LIN {X 0,Y 362.168,Z 797.832,A -85,B 0,C 180,E1 19612.506,E2 19612.506} C_VEL
LIN {X 0,Y 361.536,Z 796.314,A -85,B 0,C 180,E1 19613.999,E2 19613.999} C_VEL
LIN {X 0,Y 362.249,Z 796.809,A -85,B 0,C 180,E1 19623.883,E2 19623.883} C_VEL
LIN {X 0,Y 364.945,Z 802.489,A -85,B 0,C 180,E1 19627.878,E2 19627.878} C_VEL
LIN {X 0,Y 367.758,Z 805.063,A -85,B 0,C 180,E1 19630.43,E2 19630.43} C_VEL
LIN {X 0,Y 371.88,Z 810.734,A -85,B 0,C 180,E1 19633.506,E2 19633.506} C_VEL
LIN {X 0,Y 378.981,Z 821.207,A -85,B 0,C 180,E1 19637.693,E2 19637.693} C_VEL
LIN {X 0,Y 387.023,Z 832.702,A -85,B 0,C 180,E1 19641.464,E2 19641.464} C_VEL
LIN {X 0,Y 400.18,Z 854.108,A -85,B 0,C 180,E1 19646.784,E2 19646.784} C_VEL
LIN {X 0,Y 413.065,Z 880.296,A -85,B 0,C 180,E1 19651.645,E2 19651.645} C_VEL
LIN {X 0,Y 424.289,Z 910.677,A -85,B 0,C 180,E1 19656.18,E2 19656.18} C_VEL
LIN {X 0,Y 427.692,Z 923.118,A -85,B 0,C 180,E1 19657.818,E2 19657.818} C_VEL
LIN {X 0,Y 416.23,Z 964.506,A -85,B 0,C 180,E1 19660.322,E2 19660.322} C_VEL
LIN {X 0,Y 402.461,Z 1004.663,A -85,B 0,C 180,E1 19663.773,E2 19663.773} C_VEL
LIN {X 0,Y 388.693,Z 1040.022,A -85,B 0,C 180,E1 19668.003,E2 19668.003} C_VEL
LIN {X 0,Y 376.09,Z 1070.375,A -85,B 0,C 180,E1 19672.936,E2 19672.936} C_VEL
LIN {X 0,Y 364.901,Z 1097.162,A -85,B 0,C 180,E1 19678.824,E2 19678.824} C_VEL
LIN {X 0,Y 356.118,Z 1120.424,A -85,B 0,C 180,E1 19685.992,E2 19685.992} C_VEL
LIN {X 0,Y 351.388,Z 1136.328,A -85,B 0,C 180,E1 19693.124,E2 19693.124} C_VEL
LIN {X 0,Y 349.542,Z 1146.309,A -85,B 0,C 180,E1 19700.041,E2 19700.041} C_VEL
LIN {X 0,Y 349.172,Z 1150.432,A -85,B 0,C 180,E1 19705.033,E2 19705.033} C_VEL
LIN {X 0,Y 349.406,Z 1151.895,A -85,B 0,C 180,E1 19709.999,E2 19709.999} C_VEL
LIN {X 0,Y 349.323,Z 1149.313,A -85,B 0,C 180,E1 19717.455,E2 19717.455} C_VEL
LIN {X 0,Y 350.482,Z 1142.163,A -85,B 0,C 180,E1 19724.247,E2 19724.247} C_VEL
LIN {X 0,Y 354.503,Z 1128.114,A -85,B 0,C 180,E1 19731.898,E2 19731.898} C_VEL
LIN {X 0,Y 361.902,Z 1109.331,A -85,B 0,C 180,E1 19738.761,E2 19738.761} C_VEL
LIN {X 0,Y 372.688,Z 1085.078,A -85,B 0,C 180,E1 19745.117,E2 19745.117} C_VEL
LIN {X 0,Y 386.556,Z 1054.958,A -85,B 0,C 180,E1 19750.804,E2 19750.804} C_VEL
LIN {X 0,Y 401.988,Z 1019.714,A -85,B 0,C 180,E1 19755.578,E2 19755.578} C_VEL
LIN {X 0,Y 417.133,Z 980.614,A -85,B 0,C 180,E1 19759.349,E2 19759.349} C_VEL
LIN {X 0,Y 430.035,Z 940.71,A -85,B 0,C 180,E1 19762.083,E2 19762.083} C_VEL
LIN {X 0,Y 433.845,Z 925.859,A -85,B 0,C 180,E1 19762.938,E2 19762.938} C_VEL
LIN {X 0,Y 427.893,Z 906.219,A -85,B 0,C 180,E1 19765.929,E2 19765.929} C_VEL
LIN {X 0,Y 423.575,Z 900.256,A -85,B 0,C 180,E1 19767.396,E2 19767.396} C_VEL
LIN {X 0,Y 415.692,Z 891.837,A -85,B 0,C 180,E1 19769.971,E2 19769.971} C_VEL
LIN {X 0,Y 405.005,Z 869.047,A -85,B 0,C 180,E1 19775.094,E2 19775.094} C_VEL
LIN {X 0,Y 395.69,Z 852.613,A -85,B 0,C 180,E1 19780.05,E2 19780.05} C_VEL
LIN {X 0,Y 388.376,Z 840.695,A -85,B 0,C 180,E1 19784.924,E2 19784.924} C_VEL
LIN {X 0,Y 384.106,Z 833.994,A -85,B 0,C 180,E1 19788.805,E2 19788.805} C_VEL
LIN {X 0,Y 380.965,Z 827.944,A -85,B 0,C 180,E1 19793.437,E2 19793.437} C_VEL
LIN {X 0,Y 380.133,Z 827.154,A -85,B 0,C 180,E1 19802.281,E2 19802.281} C_VEL
LIN {X 0,Y 381.144,Z 828.782,A -85,B 0,C 180,E1 19804.693,E2 19804.693} C_VEL
LIN {X 0,Y 385.399,Z 836.304,A -85,B 0,C 180,E1 19810.307,E2 19810.307} C_VEL
LIN {X 0,Y 389.991,Z 844.13,A -85,B 0,C 180,E1 19814.191,E2 19814.191} C_VEL
LIN {X 0,Y 396.416,Z 855.261,A -85,B 0,C 180,E1 19818.472,E2 19818.472} C_VEL
LIN {X 0,Y 405.022,Z 872,A -85,B 0,C 180,E1 19823.353,E2 19823.353} C_VEL
LIN {X 0,Y 414.582,Z 895.457,A -85,B 0,C 180,E1 19828.579,E2 19828.579} C_VEL
LIN {X 0,Y 422.183,Z 920.876,A -85,B 0,C 180,E1 19833.177,E2 19833.177} C_VEL
LIN {X 0,Y 424.149,Z 932.657,A -85,B 0,C 180,E1 19834.976,E2 19834.976} C_VEL
LIN {X 0,Y 410.073,Z 973.06,A -85,B 0,C 180,E1 19838.101,E2 19838.101} C_VEL
LIN {X 0,Y 394.408,Z 1010.708,A -85,B 0,C 180,E1 19842.231,E2 19842.231} C_VEL
LIN {X 0,Y 379.532,Z 1042.173,A -85,B 0,C 180,E1 19847.015,E2 19847.015} C_VEL
LIN {X 0,Y 366.399,Z 1068.593,A -85,B 0,C 180,E1 19852.534,E2 19852.534} C_VEL
LIN {X 0,Y 354.767,Z 1091.747,A -85,B 0,C 180,E1 19859.262,E2 19859.262} C_VEL
LIN {X 0,Y 346.87,Z 1109.654,A -85,B 0,C 180,E1 19866.918,E2 19866.918} C_VEL
LIN {X 0,Y 342.767,Z 1121.009,A -85,B 0,C 180,E1 19874.663,E2 19874.663} C_VEL
LIN {X 0,Y 341.278,Z 1126.553,A -85,B 0,C 180,E1 19882.368,E2 19882.368} C_VEL
LIN {X 0,Y 341.472,Z 1126.707,A -85,B 0,C 180,E1 19890.001,E2 19890.001} C_VEL
LIN {X 0,Y 342.066,Z 1122.521,A -85,B 0,C 180,E1 19896.548,E2 19896.548} C_VEL
LIN {X 0,Y 344.669,Z 1112.858,A -85,B 0,C 180,E1 19903.955,E2 19903.955} C_VEL
LIN {X 0,Y 350.349,Z 1097.245,A -85,B 0,C 180,E1 19911.397,E2 19911.397} C_VEL
LIN {X 0,Y 360.014,Z 1075.116,A -85,B 0,C 180,E1 19918.521,E2 19918.521} C_VEL
LIN {X 0,Y 373.042,Z 1046.772,A -85,B 0,C 180,E1 19924.903,E2 19924.903} C_VEL
LIN {X 0,Y 387.331,Z 1014.182,A -85,B 0,C 180,E1 19930.139,E2 19930.139} C_VEL
LIN {X 0,Y 401.157,Z 979.377,A -85,B 0,C 180,E1 19934.184,E2 19934.184} C_VEL
LIN {X 0,Y 413.904,Z 941.564,A -85,B 0,C 180,E1 19937.419,E2 19937.419} C_VEL
LIN {X 0,Y 417.932,Z 926.539,A -85,B 0,C 180,E1 19938.504,E2 19938.504} C_VEL
LIN {X 0,Y 410.386,Z 897.331,A -85,B 0,C 180,E1 19942.987,E2 19942.987} C_VEL
LIN {X 0,Y 400.227,Z 871.059,A -85,B 0,C 180,E1 19947.767,E2 19947.767} C_VEL
LIN {X 0,Y 388.953,Z 848.616,A -85,B 0,C 180,E1 19952.842,E2 19952.842} C_VEL
LIN {X 0,Y 378.74,Z 831.473,A -85,B 0,C 180,E1 19957.951,E2 19957.951} C_VEL
LIN {X 0,Y 369.947,Z 818.286,A -85,B 0,C 180,E1 19963.385,E2 19963.385} C_VEL
LIN {X 0,Y 365.888,Z 812.166,A -85,B 0,C 180,E1 19966.717,E2 19966.717} C_VEL
LIN {X 0,Y 361.027,Z 805.323,A -85,B 0,C 180,E1 19972.86,E2 19972.86} C_VEL
LIN {X 0,Y 360.12,Z 803.979,A -85,B 0,C 180,E1 19975.183,E2 19975.183} C_VEL
LIN {X 0,Y 361.146,Z 804.69,A -85,B 0,C 180,E1 19983.669,E2 19983.669} C_VEL
LIN {X 0,Y 364.275,Z 810.621,A -85,B 0,C 180,E1 19988.193,E2 19988.193} C_VEL
LIN {X 0,Y 366.418,Z 812.851,A -85,B 0,C 180,E1 19990.164,E2 19990.164} C_VEL
LIN {X 0,Y 371.827,Z 820.887,A -85,B 0,C 180,E1 19994.257,E2 19994.257} C_VEL
LIN {X 0,Y 377.543,Z 829.283,A -85,B 0,C 180,E1 19997.612,E2 19997.612} C_VEL
LIN {X 0,Y 385.804,Z 841.914,A -85,B 0,C 180,E1 20001.686,E2 20001.686} C_VEL
LIN {X 0,Y 397.536,Z 862.222,A -85,B 0,C 180,E1 20006.672,E2 20006.672} C_VEL
LIN {X 0,Y 408.791,Z 885.918,A -85,B 0,C 180,E1 20011.156,E2 20011.156} C_VEL
LIN {X 0,Y 419.34,Z 916.182,A -85,B 0,C 180,E1 20015.795,E2 20015.795} C_VEL
LIN {X 0,Y 421.555,Z 927.264,A -85,B 0,C 180,E1 20017.21,E2 20017.21} C_VEL
LIN {X 0,Y 410.01,Z 967.1,A -85,B 0,C 180,E1 20019.709,E2 20019.709} C_VEL
LIN {X 0,Y 396.083,Z 1006.299,A -85,B 0,C 180,E1 20023.142,E2 20023.142} C_VEL
LIN {X 0,Y 381.298,Z 1042.819,A -85,B 0,C 180,E1 20027.643,E2 20027.643} C_VEL
LIN {X 0,Y 367.774,Z 1073.95,A -85,B 0,C 180,E1 20032.952,E2 20032.952} C_VEL
LIN {X 0,Y 356.83,Z 1099.215,A -85,B 0,C 180,E1 20038.821,E2 20038.821} C_VEL
LIN {X 0,Y 348.628,Z 1120.215,A -85,B 0,C 180,E1 20045.507,E2 20045.507} C_VEL
LIN {X 0,Y 343.368,Z 1137.166,A -85,B 0,C 180,E1 20053.377,E2 20053.377} C_VEL
LIN {X 0,Y 341.653,Z 1145.995,A -85,B 0,C 180,E1 20059.808,E2 20059.808} C_VEL
LIN {X 0,Y 341.284,Z 1150.137,A -85,B 0,C 180,E1 20064.918,E2 20064.918} C_VEL
LIN {X 0,Y 341.507,Z 1151.61,A -85,B 0,C 180,E1 20069.999,E2 20069.999} C_VEL
LIN {X 0,Y 341.426,Z 1149.049,A -85,B 0,C 180,E1 20077.629,E2 20077.629} C_VEL
LIN {X 0,Y 342.51,Z 1142.66,A -85,B 0,C 180,E1 20083.981,E2 20083.981} C_VEL
LIN {X 0,Y 345.94,Z 1130.613,A -85,B 0,C 180,E1 20091.121,E2 20091.121} C_VEL
LIN {X 0,Y 353.398,Z 1112.237,A -85,B 0,C 180,E1 20098.42,E2 20098.42} C_VEL
LIN {X 0,Y 365.132,Z 1086.928,A -85,B 0,C 180,E1 20105.406,E2 20105.406} C_VEL
LIN {X 0,Y 380.108,Z 1055.581,A -85,B 0,C 180,E1 20111.488,E2 20111.488} C_VEL
LIN {X 0,Y 396.368,Z 1019.642,A -85,B 0,C 180,E1 20116.413,E2 20116.413} C_VEL
LIN {X 0,Y 412.043,Z 980.377,A -85,B 0,C 180,E1 20120.214,E2 20120.214} C_VEL
LIN {X 0,Y 425.19,Z 940.845,A -85,B 0,C 180,E1 20122.925,E2 20122.925} C_VEL
LIN {X 0,Y 428.283,Z 929.273,A -85,B 0,C 180,E1 20123.606,E2 20123.606} C_VEL
LIN {X 0,Y 420.043,Z 902.49,A -85,B 0,C 180,E1 20127.962,E2 20127.962} C_VEL
LIN {X 0,Y 415.692,Z 891.837,A -85,B 0,C 180,E1 20129.971,E2 20129.971} C_VEL
LIN {X 0,Y 411.436,Z 886.846,A -85,B 0,C 180,E1 20131.549,E2 20131.549} C_VEL
LIN {X 0,Y 404.486,Z 881.278,A -85,B 0,C 180,E1 20134.056,E2 20134.056} C_VEL
LIN {X 0,Y 403.94,Z 880.243,A -85,B 0,C 180,E1 20134.322,E2 20134.322} C_VEL
LIN {X 0,Y 393.864,Z 860.717,A -85,B 0,C 180,E1 20139.954,E2 20139.954} C_VEL
LIN {X 0,Y 386.147,Z 847.843,A -85,B 0,C 180,E1 20145.415,E2 20145.415} C_VEL
LIN {X 0,Y 382.343,Z 841.592,A -85,B 0,C 180,E1 20149.041,E2 20149.041} C_VEL
LIN {X 0,Y 378.986,Z 835.151,A -85,B 0,C 180,E1 20154.64,E2 20154.64} C_VEL
LIN {X 0,Y 379.367,Z 835.251,A -85,B 0,C 180,E1 20163.857,E2 20163.857} C_VEL
LIN {X 0,Y 382.515,Z 841.74,A -85,B 0,C 180,E1 20168.879,E2 20168.879} C_VEL
LIN {X 0,Y 387.602,Z 851.333,A -85,B 0,C 180,E1 20173.863,E2 20173.863} C_VEL
LIN {X 0,Y 393.503,Z 862.183,A -85,B 0,C 180,E1 20178.108,E2 20178.108} C_VEL
LIN {X 0,Y 401.875,Z 879.654,A -85,B 0,C 180,E1 20183.254,E2 20183.254} C_VEL
LIN {X 0,Y 410.458,Z 901.841,A -85,B 0,C 180,E1 20188.263,E2 20188.263} C_VEL
LIN {X 0,Y 417.611,Z 928.524,A -85,B 0,C 180,E1 20193.179,E2 20193.179} C_VEL
LIN {X 0,Y 418.331,Z 936.224,A -85,B 0,C 180,E1 20194.321,E2 20194.321} C_VEL
LIN {X 0,Y 404.003,Z 975.78,A -85,B 0,C 180,E1 20197.458,E2 20197.458} C_VEL
LIN {X 0,Y 388.289,Z 1012.281,A -85,B 0,C 180,E1 20201.538,E2 20201.538} C_VEL
LIN {X 0,Y 372.079,Z 1045.221,A -85,B 0,C 180,E1 20206.684,E2 20206.684} C_VEL
LIN {X 0,Y 357.973,Z 1072.305,A -85,B 0,C 180,E1 20212.643,E2 20212.643} C_VEL
LIN {X 0,Y 346.862,Z 1093.638,A -85,B 0,C 180,E1 20219.212,E2 20219.212} C_VEL
LIN {X 0,Y 339.389,Z 1109.871,A -85,B 0,C 180,E1 20226.379,E2 20226.379} C_VEL
LIN {X 0,Y 334.988,Z 1121.246,A -85,B 0,C 180,E1 20234.298,E2 20234.298} C_VEL
LIN {X 0,Y 333.385,Z 1126.82,A -85,B 0,C 180,E1 20242.186,E2 20242.186} C_VEL
LIN {X 0,Y 333.328,Z 1127.532,A -85,B 0,C 180,E1 20247.403,E2 20247.403} C_VEL
LIN {X 0,Y 333.695,Z 1125.898,A -85,B 0,C 180,E1 20252.597,E2 20252.597} C_VEL
LIN {X 0,Y 334.796,Z 1120.388,A -85,B 0,C 180,E1 20259.091,E2 20259.091} C_VEL
LIN {X 0,Y 338.283,Z 1109.482,A -85,B 0,C 180,E1 20266.443,E2 20266.443} C_VEL
LIN {X 0,Y 345.277,Z 1092.289,A -85,B 0,C 180,E1 20273.882,E2 20273.882} C_VEL
LIN {X 0,Y 355.746,Z 1069.725,A -85,B 0,C 180,E1 20280.647,E2 20280.647} C_VEL
LIN {X 0,Y 368.456,Z 1043,A -85,B 0,C 180,E1 20286.402,E2 20286.402} C_VEL
LIN {X 0,Y 383.057,Z 1010.649,A -85,B 0,C 180,E1 20291.457,E2 20291.457} C_VEL
LIN {X 0,Y 397.955,Z 973.716,A -85,B 0,C 180,E1 20295.603,E2 20295.603} C_VEL
LIN {X 0,Y 411.711,Z 932.607,A -85,B 0,C 180,E1 20298.891,E2 20298.891} C_VEL
LIN {X 0,Y 411.505,Z 926.566,A -85,B 0,C 180,E1 20299.627,E2 20299.627} C_VEL
LIN {X 0,Y 404.09,Z 897.94,A -85,B 0,C 180,E1 20304.243,E2 20304.243} C_VEL
LIN {X 0,Y 393.436,Z 870.633,A -85,B 0,C 180,E1 20309.569,E2 20309.569} C_VEL
LIN {X 0,Y 382.417,Z 849.153,A -85,B 0,C 180,E1 20314.976,E2 20314.976} C_VEL
LIN {X 0,Y 374.275,Z 835.712,A -85,B 0,C 180,E1 20319.516,E2 20319.516} C_VEL
LIN {X 0,Y 367.793,Z 825.425,A -85,B 0,C 180,E1 20324.031,E2 20324.031} C_VEL
LIN {X 0,Y 363.665,Z 818.969,A -85,B 0,C 180,E1 20327.703,E2 20327.703} C_VEL
LIN {X 0,Y 359.883,Z 812.953,A -85,B 0,C 180,E1 20333.14,E2 20333.14} C_VEL
LIN {X 0,Y 358.713,Z 811.507,A -85,B 0,C 180,E1 20337.582,E2 20337.582} C_VEL
LIN {X 0,Y 360.103,Z 812.832,A -85,B 0,C 180,E1 20343.605,E2 20343.605} C_VEL
LIN {X 0,Y 363.845,Z 818.876,A -85,B 0,C 180,E1 20348.804,E2 20348.804} C_VEL
LIN {X 0,Y 370.025,Z 828.147,A -85,B 0,C 180,E1 20353.876,E2 20353.876} C_VEL
LIN {X 0,Y 378.227,Z 840.611,A -85,B 0,C 180,E1 20358.784,E2 20358.784} C_VEL
LIN {X 0,Y 389.385,Z 859.782,A -85,B 0,C 180,E1 20364.191,E2 20364.191} C_VEL
LIN {X 0,Y 401.157,Z 883.666,A -85,B 0,C 180,E1 20369.264,E2 20369.264} C_VEL
LIN {X 0,Y 411.593,Z 912.314,A -85,B 0,C 180,E1 20374.037,E2 20374.037} C_VEL
LIN {X 0,Y 415.852,Z 929.747,A -85,B 0,C 180,E1 20376.488,E2 20376.488} C_VEL
LIN {X 0,Y 403.786,Z 969.68,A -85,B 0,C 180,E1 20379.07,E2 20379.07} C_VEL
LIN {X 0,Y 389.596,Z 1008.144,A -85,B 0,C 180,E1 20382.527,E2 20382.527} C_VEL
LIN {X 0,Y 374.466,Z 1044.278,A -85,B 0,C 180,E1 20387.079,E2 20387.079} C_VEL
LIN {X 0,Y 359.392,Z 1077.666,A -85,B 0,C 180,E1 20393.004,E2 20393.004} C_VEL
LIN {X 0,Y 347.197,Z 1104.998,A -85,B 0,C 180,E1 20399.885,E2 20399.885} C_VEL
LIN {X 0,Y 338.739,Z 1126.558,A -85,B 0,C 180,E1 20407.715,E2 20407.715} C_VEL
LIN {X 0,Y 334.81,Z 1139.995,A -85,B 0,C 180,E1 20415.035,E2 20415.035} C_VEL
LIN {X 0,Y 333.546,Z 1148.087,A -85,B 0,C 180,E1 20422.187,E2 20422.187} C_VEL
LIN {X 0,Y 333.435,Z 1150.905,A -85,B 0,C 180,E1 20427.401,E2 20427.401} C_VEL
LIN {X 0,Y 333.404,Z 1151.1,A -85,B 0,C 180,E1 20432.596,E2 20432.596} C_VEL
LIN {X 0,Y 333.647,Z 1147.89,A -85,B 0,C 180,E1 20439.119,E2 20439.119} C_VEL
LIN {X 0,Y 335.145,Z 1140.554,A -85,B 0,C 180,E1 20445.694,E2 20445.694} C_VEL
LIN {X 0,Y 340.055,Z 1126.288,A -85,B 0,C 180,E1 20453.572,E2 20453.572} C_VEL
LIN {X 0,Y 349.349,Z 1105.179,A -85,B 0,C 180,E1 20461.267,E2 20461.267} C_VEL
LIN {X 0,Y 363.057,Z 1077.643,A -85,B 0,C 180,E1 20468.187,E2 20468.187} C_VEL
LIN {X 0,Y 379.117,Z 1044.881,A -85,B 0,C 180,E1 20473.963,E2 20473.963} C_VEL
LIN {X 0,Y 395.082,Z 1009.645,A -85,B 0,C 180,E1 20478.364,E2 20478.364} C_VEL
LIN {X 0,Y 409.577,Z 973.339,A -85,B 0,C 180,E1 20481.627,E2 20481.627} C_VEL
LIN {X 0,Y 422.829,Z 932.79,A -85,B 0,C 180,E1 20484.272,E2 20484.272} C_VEL
LIN {X 0,Y 414.989,Z 906.692,A -85,B 0,C 180,E1 20488.677,E2 20488.677} C_VEL
LIN {X 0,Y 404.705,Z 881.627,A -85,B 0,C 180,E1 20493.956,E2 20493.956} C_VEL
LIN {X 0,Y 403.94,Z 880.243,A -85,B 0,C 180,E1 20494.322,E2 20494.322} C_VEL
LIN {X 0,Y 400.075,Z 875.927,A -85,B 0,C 180,E1 20495.995,E2 20495.995} C_VEL
LIN {X 0,Y 393.13,Z 871.803,A -85,B 0,C 180,E1 20498.985,E2 20498.985} C_VEL
LIN {X 0,Y 384.724,Z 856.032,A -85,B 0,C 180,E1 20505.069,E2 20505.069} C_VEL
LIN {X 0,Y 380.382,Z 849.039,A -85,B 0,C 180,E1 20509.418,E2 20509.418} C_VEL
LIN {X 0,Y 377.669,Z 842.974,A -85,B 0,C 180,E1 20514.264,E2 20514.264} C_VEL
LIN {X 0,Y 377.788,Z 843.047,A -85,B 0,C 180,E1 20523.73,E2 20523.73} C_VEL
LIN {X 0,Y 380.727,Z 849.492,A -85,B 0,C 180,E1 20528.921,E2 20528.921} C_VEL
LIN {X 0,Y 387.257,Z 861.984,A -85,B 0,C 180,E1 20535.2,E2 20535.2} C_VEL
LIN {X 0,Y 395.349,Z 879.25,A -85,B 0,C 180,E1 20540.998,E2 20540.998} C_VEL
LIN {X 0,Y 403.722,Z 900.712,A -85,B 0,C 180,E1 20546.359,E2 20546.359} C_VEL
LIN {X 0,Y 410.328,Z 923.987,A -85,B 0,C 180,E1 20551.034,E2 20551.034} C_VEL
LIN {X 0,Y 412.849,Z 938.974,A -85,B 0,C 180,E1 20553.592,E2 20553.592} C_VEL
LIN {X 0,Y 398.879,Z 976.352,A -85,B 0,C 180,E1 20556.595,E2 20556.595} C_VEL
LIN {X 0,Y 382.928,Z 1012.308,A -85,B 0,C 180,E1 20560.624,E2 20560.624} C_VEL
LIN {X 0,Y 366.202,Z 1045.309,A -85,B 0,C 180,E1 20565.81,E2 20565.81} C_VEL
LIN {X 0,Y 352.17,Z 1071.253,A -85,B 0,C 180,E1 20571.527,E2 20571.527} C_VEL
LIN {X 0,Y 340.775,Z 1092.108,A -85,B 0,C 180,E1 20577.853,E2 20577.853} C_VEL
LIN {X 0,Y 331.938,Z 1110.085,A -85,B 0,C 180,E1 20585.815,E2 20585.815} C_VEL
LIN {X 0,Y 327.249,Z 1121.482,A -85,B 0,C 180,E1 20593.917,E2 20593.917} C_VEL
LIN {X 0,Y 325.493,Z 1127.087,A -85,B 0,C 180,E1 20601.996,E2 20601.996} C_VEL
LIN {X 0,Y 325.43,Z 1127.819,A -85,B 0,C 180,E1 20607.34,E2 20607.34} C_VEL
LIN {X 0,Y 325.813,Z 1126.206,A -85,B 0,C 180,E1 20612.66,E2 20612.66} C_VEL
LIN {X 0,Y 326.97,Z 1120.719,A -85,B 0,C 180,E1 20619.31,E2 20619.31} C_VEL
LIN {X 0,Y 330.453,Z 1110.344,A -85,B 0,C 180,E1 20626.539,E2 20626.539} C_VEL
LIN {X 0,Y 337.172,Z 1094.37,A -85,B 0,C 180,E1 20633.79,E2 20633.79} C_VEL
LIN {X 0,Y 347.161,Z 1073.675,A -85,B 0,C 180,E1 20640.4,E2 20640.4} C_VEL
LIN {X 0,Y 360.579,Z 1046.711,A -85,B 0,C 180,E1 20646.552,E2 20646.552} C_VEL
LIN {X 0,Y 376.254,Z 1013.188,A -85,B 0,C 180,E1 20651.994,E2 20651.994} C_VEL
LIN {X 0,Y 391.949,Z 975.567,A -85,B 0,C 180,E1 20656.306,E2 20656.306} C_VEL
LIN {X 0,Y 405.592,Z 936.216,A -85,B 0,C 180,E1 20659.533,E2 20659.533} C_VEL
LIN {X 0,Y 405.888,Z 930.287,A -85,B 0,C 180,E1 20660.23,E2 20660.23} C_VEL
LIN {X 0,Y 399.275,Z 903.126,A -85,B 0,C 180,E1 20664.752,E2 20664.752} C_VEL
LIN {X 0,Y 389.421,Z 876.566,A -85,B 0,C 180,E1 20670.061,E2 20670.061} C_VEL
LIN {X 0,Y 379.183,Z 855.426,A -85,B 0,C 180,E1 20675.554,E2 20675.554} C_VEL
LIN {X 0,Y 370.32,Z 839.719,A -85,B 0,C 180,E1 20681.027,E2 20681.027} C_VEL
LIN {X 0,Y 365.445,Z 832.455,A -85,B 0,C 180,E1 20684.65,E2 20684.65} C_VEL
LIN {X 0,Y 361.967,Z 826.507,A -85,B 0,C 180,E1 20688.205,E2 20688.205} C_VEL
LIN {X 0,Y 358.567,Z 820.126,A -85,B 0,C 180,E1 20693.646,E2 20693.646} C_VEL
LIN {X 0,Y 358.803,Z 820.091,A -85,B 0,C 180,E1 20703.164,E2 20703.164} C_VEL
LIN {X 0,Y 362.094,Z 826.331,A -85,B 0,C 180,E1 20708.243,E2 20708.243} C_VEL
LIN {X 0,Y 363.768,Z 828.917,A -85,B 0,C 180,E1 20709.937,E2 20709.937} C_VEL
LIN {X 0,Y 368.356,Z 835.989,A -85,B 0,C 180,E1 20713.713,E2 20713.713} C_VEL
LIN {X 0,Y 376.027,Z 848.137,A -85,B 0,C 180,E1 20718.518,E2 20718.518} C_VEL
LIN {X 0,Y 386.853,Z 867.538,A -85,B 0,C 180,E1 20724.054,E2 20724.054} C_VEL
LIN {X 0,Y 397.426,Z 890.611,A -85,B 0,C 180,E1 20729.01,E2 20729.01} C_VEL
LIN {X 0,Y 407.103,Z 919.151,A -85,B 0,C 180,E1 20733.823,E2 20733.823} C_VEL
LIN {X 0,Y 410.257,Z 931.658,A -85,B 0,C 180,E1 20735.696,E2 20735.696} C_VEL
LIN {X 0,Y 397.025,Z 973.907,A -85,B 0,C 180,E1 20738.536,E2 20738.536} C_VEL
LIN {X 0,Y 383.326,Z 1009.53,A -85,B 0,C 180,E1 20741.841,E2 20741.841} C_VEL
LIN {X 0,Y 368.52,Z 1043.8,A -85,B 0,C 180,E1 20746.213,E2 20746.213} C_VEL
LIN {X 0,Y 352.898,Z 1077.24,A -85,B 0,C 180,E1 20752.205,E2 20752.205} C_VEL
LIN {X 0,Y 340.007,Z 1104.835,A -85,B 0,C 180,E1 20759.261,E2 20759.261} C_VEL
LIN {X 0,Y 331.227,Z 1126.198,A -85,B 0,C 180,E1 20767.182,E2 20767.182} C_VEL
LIN {X 0,Y 326.845,Z 1140.502,A -85,B 0,C 180,E1 20775.242,E2 20775.242} C_VEL
LIN {X 0,Y 325.65,Z 1147.783,A -85,B 0,C 180,E1 20781.996,E2 20781.996} C_VEL
LIN {X 0,Y 325.529,Z 1150.612,A -85,B 0,C 180,E1 20787.338,E2 20787.338} C_VEL
LIN {X 0,Y 325.5,Z 1150.823,A -85,B 0,C 180,E1 20792.659,E2 20792.659} C_VEL
LIN {X 0,Y 325.785,Z 1147.626,A -85,B 0,C 180,E1 20799.341,E2 20799.341} C_VEL
LIN {X 0,Y 327.405,Z 1140.314,A -85,B 0,C 180,E1 20806.075,E2 20806.075} C_VEL
LIN {X 0,Y 332.593,Z 1126.067,A -85,B 0,C 180,E1 20814.135,E2 20814.135} C_VEL
LIN {X 0,Y 342.411,Z 1104.986,A -85,B 0,C 180,E1 20821.975,E2 20821.975} C_VEL
LIN {X 0,Y 356.059,Z 1078.611,A -85,B 0,C 180,E1 20828.748,E2 20828.748} C_VEL
LIN {X 0,Y 371.239,Z 1048.787,A -85,B 0,C 180,E1 20834.21,E2 20834.21} C_VEL
LIN {X 0,Y 387.036,Z 1015.824,A -85,B 0,C 180,E1 20838.564,E2 20838.564} C_VEL
LIN {X 0,Y 402.968,Z 977.945,A -85,B 0,C 180,E1 20842.168,E2 20842.168} C_VEL
LIN {X 0,Y 417.168,Z 935.697,A -85,B 0,C 180,E1 20845.043,E2 20845.043} C_VEL
LIN {X 0,Y 409.307,Z 908.802,A -85,B 0,C 180,E1 20849.81,E2 20849.81} C_VEL
LIN {X 0,Y 400.089,Z 885.921,A -85,B 0,C 180,E1 20854.924,E2 20854.924} C_VEL
LIN {X 0,Y 393.13,Z 871.803,A -85,B 0,C 180,E1 20858.985,E2 20858.985} C_VEL
LIN {X 0,Y 383.944,Z 866.755,A -85,B 0,C 180,E1 20863.942,E2 20863.942} C_VEL
LIN {X 0,Y 378.689,Z 856.9,A -85,B 0,C 180,E1 20869.225,E2 20869.225} C_VEL
LIN {X 0,Y 375.718,Z 850.567,A -85,B 0,C 180,E1 20874.812,E2 20874.812} C_VEL
LIN {X 0,Y 375.909,Z 850.766,A -85,B 0,C 180,E1 20883.604,E2 20883.604} C_VEL
LIN {X 0,Y 379.379,Z 859.105,A -85,B 0,C 180,E1 20889.748,E2 20889.748} C_VEL
LIN {X 0,Y 384.502,Z 869.078,A -85,B 0,C 180,E1 20894.874,E2 20894.874} C_VEL
LIN {X 0,Y 392.77,Z 888.014,A -85,B 0,C 180,E1 20901.219,E2 20901.219} C_VEL
LIN {X 0,Y 400.164,Z 908.969,A -85,B 0,C 180,E1 20906.476,E2 20906.476} C_VEL
LIN {X 0,Y 406.245,Z 933.446,A -85,B 0,C 180,E1 20911.381,E2 20911.381} C_VEL
LIN {X 0,Y 407.489,Z 941.696,A -85,B 0,C 180,E1 20912.85,E2 20912.85} C_VEL
LIN {X 0,Y 393.181,Z 978.428,A -85,B 0,C 180,E1 20915.853,E2 20915.853} C_VEL
LIN {X 0,Y 376.512,Z 1014.676,A -85,B 0,C 180,E1 20920,E2 20920} C_VEL
LIN {X 0,Y 359.419,Z 1047.186,A -85,B 0,C 180,E1 20925.228,E2 20925.228} C_VEL
LIN {X 0,Y 343.737,Z 1074.964,A -85,B 0,C 180,E1 20931.616,E2 20931.616} C_VEL
LIN {X 0,Y 331.918,Z 1095.712,A -85,B 0,C 180,E1 20938.431,E2 20938.431} C_VEL
LIN {X 0,Y 323.933,Z 1111.426,A -85,B 0,C 180,E1 20945.911,E2 20945.911} C_VEL
LIN {X 0,Y 319.493,Z 1121.72,A -85,B 0,C 180,E1 20953.516,E2 20953.516} C_VEL
LIN {X 0,Y 317.602,Z 1127.355,A -85,B 0,C 180,E1 20961.795,E2 20961.795} C_VEL
LIN {X 0,Y 317.549,Z 1128.047,A -85,B 0,C 180,E1 20967.732,E2 20967.732} C_VEL
LIN {X 0,Y 317.994,Z 1125.865,A -85,B 0,C 180,E1 20973.785,E2 20973.785} C_VEL
LIN {X 0,Y 319.578,Z 1119.538,A -85,B 0,C 180,E1 20980.904,E2 20980.904} C_VEL
LIN {X 0,Y 323.845,Z 1108.074,A -85,B 0,C 180,E1 20988.36,E2 20988.36} C_VEL
LIN {X 0,Y 331.552,Z 1091.372,A -85,B 0,C 180,E1 20995.658,E2 20995.658} C_VEL
LIN {X 0,Y 343.983,Z 1066.921,A -85,B 0,C 180,E1 21002.983,E2 21002.983} C_VEL
LIN {X 0,Y 359.118,Z 1037.325,A -85,B 0,C 180,E1 21009.138,E2 21009.138} C_VEL
LIN {X 0,Y 374.731,Z 1004.024,A -85,B 0,C 180,E1 21014.077,E2 21014.077} C_VEL
LIN {X 0,Y 389.608,Z 968.224,A -85,B 0,C 180,E1 21017.884,E2 21017.884} C_VEL
LIN {X 0,Y 400.512,Z 935.803,A -85,B 0,C 180,E1 21020.539,E2 21020.539} C_VEL
LIN {X 0,Y 394.377,Z 908.239,A -85,B 0,C 180,E1 21025.256,E2 21025.256} C_VEL
LIN {X 0,Y 385.437,Z 882.576,A -85,B 0,C 180,E1 21030.545,E2 21030.545} C_VEL
LIN {X 0,Y 376.01,Z 862.069,A -85,B 0,C 180,E1 21035.99,E2 21035.99} C_VEL
LIN {X 0,Y 367.793,Z 846.8,A -85,B 0,C 180,E1 21041.459,E2 21041.459} C_VEL
LIN {X 0,Y 363.39,Z 839.781,A -85,B 0,C 180,E1 21045.056,E2 21045.056} C_VEL
LIN {X 0,Y 360.048,Z 833.919,A -85,B 0,C 180,E1 21048.652,E2 21048.652} C_VEL
LIN {X 0,Y 357.095,Z 827.473,A -85,B 0,C 180,E1 21054.534,E2 21054.534} C_VEL
LIN {X 0,Y 357.586,Z 828.165,A -85,B 0,C 180,E1 21063.099,E2 21063.099} C_VEL
LIN {X 0,Y 361.265,Z 834.443,A -85,B 0,C 180,E1 21068.716,E2 21068.716} C_VEL
LIN {X 0,Y 366.619,Z 843.923,A -85,B 0,C 180,E1 21073.627,E2 21073.627} C_VEL
LIN {X 0,Y 373.705,Z 855.774,A -85,B 0,C 180,E1 21078.332,E2 21078.332} C_VEL
LIN {X 0,Y 383.997,Z 875.148,A -85,B 0,C 180,E1 21083.924,E2 21083.924} C_VEL
LIN {X 0,Y 394.603,Z 900.168,A -85,B 0,C 180,E1 21089.238,E2 21089.238} C_VEL
LIN {X 0,Y 403.088,Z 928.393,A -85,B 0,C 180,E1 21094.025,E2 21094.025} C_VEL
LIN {X 0,Y 404.362,Z 935.699,A -85,B 0,C 180,E1 21095.06,E2 21095.06} C_VEL
LIN {X 0,Y 390.477,Z 977.703,A -85,B 0,C 180,E1 21097.955,E2 21097.955} C_VEL
LIN {X 0,Y 374.936,Z 1016.114,A -85,B 0,C 180,E1 21101.724,E2 21101.724} C_VEL
LIN {X 0,Y 360.049,Z 1048.704,A -85,B 0,C 180,E1 21106.17,E2 21106.17} C_VEL
LIN {X 0,Y 345.317,Z 1078.975,A -85,B 0,C 180,E1 21111.861,E2 21111.861} C_VEL
LIN {X 0,Y 332.941,Z 1104.439,A -85,B 0,C 180,E1 21118.535,E2 21118.535} C_VEL
LIN {X 0,Y 323.711,Z 1125.836,A -85,B 0,C 180,E1 21126.621,E2 21126.621} C_VEL
LIN {X 0,Y 319.048,Z 1140.206,A -85,B 0,C 180,E1 21134.899,E2 21134.899} C_VEL
LIN {X 0,Y 317.774,Z 1147.48,A -85,B 0,C 180,E1 21141.797,E2 21141.797} C_VEL
LIN {X 0,Y 317.637,Z 1150.318,A -85,B 0,C 180,E1 21147.272,E2 21147.272} C_VEL
LIN {X 0,Y 317.614,Z 1150.546,A -85,B 0,C 180,E1 21152.725,E2 21152.725} C_VEL
LIN {X 0,Y 317.921,Z 1147.363,A -85,B 0,C 180,E1 21159.575,E2 21159.575} C_VEL
LIN {X 0,Y 319.648,Z 1140.073,A -85,B 0,C 180,E1 21166.476,E2 21166.476} C_VEL
LIN {X 0,Y 325.181,Z 1125.847,A -85,B 0,C 180,E1 21174.721,E2 21174.721} C_VEL
LIN {X 0,Y 335.486,Z 1104.791,A -85,B 0,C 180,E1 21182.716,E2 21182.716} C_VEL
LIN {X 0,Y 350.026,Z 1078.004,A -85,B 0,C 180,E1 21189.681,E2 21189.681} C_VEL
LIN {X 0,Y 365.95,Z 1047.779,A -85,B 0,C 180,E1 21195.235,E2 21195.235} C_VEL
LIN {X 0,Y 382.652,Z 1013.743,A -85,B 0,C 180,E1 21199.697,E2 21199.697} C_VEL
LIN {X 0,Y 398.699,Z 976.454,A -85,B 0,C 180,E1 21203.191,E2 21203.191} C_VEL
LIN {X 0,Y 411.66,Z 939.215,A -85,B 0,C 180,E1 21205.731,E2 21205.731} C_VEL
LIN {X 0,Y 404.8,Z 914.149,A -85,B 0,C 180,E1 21210.341,E2 21210.341} C_VEL
LIN {X 0,Y 395.753,Z 890.567,A -85,B 0,C 180,E1 21215.774,E2 21215.774} C_VEL
LIN {X 0,Y 387.603,Z 873.8,A -85,B 0,C 180,E1 21221.068,E2 21221.068} C_VEL
LIN {X 0,Y 383.944,Z 866.755,A -85,B 0,C 180,E1 21223.942,E2 21223.942} C_VEL
LIN {X 0,Y 381.372,Z 864.663,A -85,B 0,C 180,E1 21225.827,E2 21225.827} C_VEL
LIN {X 0,Y 376.903,Z 864.655,A -85,B 0,C 180,E1 21229.103,E2 21229.103} C_VEL
LIN {X 0,Y 373.882,Z 858.254,A -85,B 0,C 180,E1 21234.787,E2 21234.787} C_VEL
LIN {X 0,Y 373.989,Z 858.474,A -85,B 0,C 180,E1 21243.478,E2 21243.478} C_VEL
LIN {X 0,Y 377.041,Z 866.741,A -85,B 0,C 180,E1 21249.663,E2 21249.663} C_VEL
LIN {X 0,Y 381.445,Z 875.681,A -85,B 0,C 180,E1 21254.336,E2 21254.336} C_VEL
LIN {X 0,Y 388.611,Z 893.258,A -85,B 0,C 180,E1 21260.485,E2 21260.485} C_VEL
LIN {X 0,Y 395.385,Z 913.596,A -85,B 0,C 180,E1 21265.767,E2 21265.767} C_VEL
LIN {X 0,Y 400.908,Z 937.73,A -85,B 0,C 180,E1 21270.793,E2 21270.793} C_VEL
LIN {X 0,Y 401.54,Z 946.214,A -85,B 0,C 180,E1 21272.206,E2 21272.206} C_VEL
LIN {X 0,Y 385.131,Z 986.111,A -85,B 0,C 180,E1 21275.659,E2 21275.659} C_VEL
LIN {X 0,Y 368.597,Z 1019.893,A -85,B 0,C 180,E1 21279.767,E2 21279.767} C_VEL
LIN {X 0,Y 352.391,Z 1049.424,A -85,B 0,C 180,E1 21284.723,E2 21284.723} C_VEL
LIN {X 0,Y 336.663,Z 1076.283,A -85,B 0,C 180,E1 21291.071,E2 21291.071} C_VEL
LIN {X 0,Y 324.003,Z 1097.604,A -85,B 0,C 180,E1 21298.355,E2 21298.355} C_VEL
LIN {X 0,Y 315.734,Z 1113.1,A -85,B 0,C 180,E1 21306.221,E2 21306.221} C_VEL
LIN {X 0,Y 311.753,Z 1121.958,A -85,B 0,C 180,E1 21313.094,E2 21313.094} C_VEL
LIN {X 0,Y 310.111,Z 1126.345,A -85,B 0,C 180,E1 21318.762,E2 21318.762} C_VEL
LIN {X 0,Y 309.604,Z 1128.301,A -85,B 0,C 180,E1 21324.4,E2 21324.4} C_VEL
LIN {X 0,Y 309.907,Z 1127.894,A -85,B 0,C 180,E1 21330.002,E2 21330.002} C_VEL
LIN {X 0,Y 310.597,Z 1123.987,A -85,B 0,C 180,E1 21336.988,E2 21336.988} C_VEL
LIN {X 0,Y 313.61,Z 1114.945,A -85,B 0,C 180,E1 21344.941,E2 21344.941} C_VEL
LIN {X 0,Y 320.823,Z 1098.756,A -85,B 0,C 180,E1 21353.498,E2 21353.498} C_VEL
LIN {X 0,Y 332.857,Z 1075.713,A -85,B 0,C 180,E1 21361.473,E2 21361.473} C_VEL
LIN {X 0,Y 347.532,Z 1048.253,A -85,B 0,C 180,E1 21367.997,E2 21367.997} C_VEL
LIN {X 0,Y 363.178,Z 1017.074,A -85,B 0,C 180,E1 21373.255,E2 21373.255} C_VEL
LIN {X 0,Y 378.531,Z 983.123,A -85,B 0,C 180,E1 21377.377,E2 21377.377} C_VEL
LIN {X 0,Y 393.204,Z 944.516,A -85,B 0,C 180,E1 21380.789,E2 21380.789} C_VEL
LIN {X 0,Y 394.679,Z 938.576,A -85,B 0,C 180,E1 21381.308,E2 21381.308} C_VEL
LIN {X 0,Y 389.161,Z 912.175,A -85,B 0,C 180,E1 21386.002,E2 21386.002} C_VEL
LIN {X 0,Y 381.104,Z 887.648,A -85,B 0,C 180,E1 21391.258,E2 21391.258} C_VEL
LIN {X 0,Y 372.296,Z 867.626,A -85,B 0,C 180,E1 21396.767,E2 21396.767} C_VEL
LIN {X 0,Y 364.979,Z 853.542,A -85,B 0,C 180,E1 21402.069,E2 21402.069} C_VEL
LIN {X 0,Y 361.019,Z 846.766,A -85,B 0,C 180,E1 21405.606,E2 21405.606} C_VEL
LIN {X 0,Y 358.456,Z 841.641,A -85,B 0,C 180,E1 21408.736,E2 21408.736} C_VEL
LIN {X 0,Y 355.425,Z 835.16,A -85,B 0,C 180,E1 21415.119,E2 21415.119} C_VEL
LIN {X 0,Y 356.075,Z 835.968,A -85,B 0,C 180,E1 21422.96,E2 21422.96} C_VEL
LIN {X 0,Y 360.19,Z 843.854,A -85,B 0,C 180,E1 21429.351,E2 21429.351} C_VEL
LIN {X 0,Y 364.565,Z 851.493,A -85,B 0,C 180,E1 21433.4,E2 21433.4} C_VEL
LIN {X 0,Y 371.208,Z 863.164,A -85,B 0,C 180,E1 21438.076,E2 21438.076} C_VEL
LIN {X 0,Y 380.594,Z 881.85,A -85,B 0,C 180,E1 21443.533,E2 21443.533} C_VEL
LIN {X 0,Y 389.925,Z 905.205,A -85,B 0,C 180,E1 21448.649,E2 21448.649} C_VEL
LIN {X 0,Y 397.752,Z 932.489,A -85,B 0,C 180,E1 21453.415,E2 21453.415} C_VEL
LIN {X 0,Y 398.412,Z 939.292,A -85,B 0,C 180,E1 21454.36,E2 21454.36} C_VEL
LIN {X 0,Y 384.435,Z 979.974,A -85,B 0,C 180,E1 21457.251,E2 21457.251} C_VEL
LIN {X 0,Y 368.316,Z 1018.482,A -85,B 0,C 180,E1 21461.113,E2 21461.113} C_VEL
LIN {X 0,Y 351.615,Z 1053.61,A -85,B 0,C 180,E1 21466.136,E2 21466.136} C_VEL
LIN {X 0,Y 336.757,Z 1082.717,A -85,B 0,C 180,E1 21471.975,E2 21471.975} C_VEL
LIN {X 0,Y 324.972,Z 1106.056,A -85,B 0,C 180,E1 21478.456,E2 21478.456} C_VEL
LIN {X 0,Y 316.196,Z 1125.563,A -85,B 0,C 180,E1 21486.076,E2 21486.076} C_VEL
LIN {X 0,Y 311.273,Z 1139.873,A -85,B 0,C 180,E1 21494.512,E2 21494.512} C_VEL
LIN {X 0,Y 309.884,Z 1147.176,A -85,B 0,C 180,E1 21501.586,E2 21501.586} C_VEL
LIN {X 0,Y 309.759,Z 1150.025,A -85,B 0,C 180,E1 21507.202,E2 21507.202} C_VEL
LIN {X 0,Y 309.706,Z 1150.268,A -85,B 0,C 180,E1 21512.795,E2 21512.795} C_VEL
LIN {X 0,Y 310.035,Z 1147.098,A -85,B 0,C 180,E1 21519.82,E2 21519.82} C_VEL
LIN {X 0,Y 311.899,Z 1139.831,A -85,B 0,C 180,E1 21526.898,E2 21526.898} C_VEL
LIN {X 0,Y 317.95,Z 1125.332,A -85,B 0,C 180,E1 21535.475,E2 21535.475} C_VEL
LIN {X 0,Y 328.642,Z 1104.597,A -85,B 0,C 180,E1 21543.486,E2 21543.486} C_VEL
LIN {X 0,Y 343.542,Z 1078.284,A -85,B 0,C 180,E1 21550.449,E2 21550.449} C_VEL
LIN {X 0,Y 359.547,Z 1049.037,A -85,B 0,C 180,E1 21555.935,E2 21555.935} C_VEL
LIN {X 0,Y 376.428,Z 1015.993,A -85,B 0,C 180,E1 21560.374,E2 21560.374} C_VEL
LIN {X 0,Y 393.957,Z 976.48,A -85,B 0,C 180,E1 21564.122,E2 21564.122} C_VEL
LIN {X 0,Y 406.1,Z 942.36,A -85,B 0,C 180,E1 21566.511,E2 21566.511} C_VEL
LIN {X 0,Y 399.936,Z 918.55,A -85,B 0,C 180,E1 21571.063,E2 21571.063} C_VEL
LIN {X 0,Y 392.22,Z 897.181,A -85,B 0,C 180,E1 21576.146,E2 21576.146} C_VEL
LIN {X 0,Y 384.558,Z 880.476,A -85,B 0,C 180,E1 21581.54,E2 21581.54} C_VEL
LIN {X 0,Y 378.944,Z 869.522,A -85,B 0,C 180,E1 21586.477,E2 21586.477} C_VEL
LIN {X 0,Y 376.903,Z 864.655,A -85,B 0,C 180,E1 21589.103,E2 21589.103} C_VEL
LIN {X 0,Y 374.391,Z 866.964,A -85,B 0,C 180,E1 21590.849,E2 21590.849} C_VEL
LIN {X 0,Y 372.498,Z 868.967,A -85,B 0,C 180,E1 21592.382,E2 21592.382} C_VEL
LIN {X 0,Y 372.386,Z 868.772,A -85,B 0,C 180,E1 21592.606,E2 21592.606} C_VEL
LIN {X 0,Y 371.671,Z 865.75,A -85,B 0,C 180,E1 21595.34,E2 21595.34} C_VEL
LIN {X 0,Y 371.836,Z 866.17,A -85,B 0,C 180,E1 21603.425,E2 21603.425} C_VEL
LIN {X 0,Y 374.654,Z 874.23,A -85,B 0,C 180,E1 21609.506,E2 21609.506} C_VEL
LIN {X 0,Y 378.808,Z 883.74,A -85,B 0,C 180,E1 21614.438,E2 21614.438} C_VEL
LIN {X 0,Y 385.583,Z 901.567,A -85,B 0,C 180,E1 21620.653,E2 21620.653} C_VEL
LIN {X 0,Y 391.292,Z 920.623,A -85,B 0,C 180,E1 21625.62,E2 21625.62} C_VEL
LIN {X 0,Y 395.901,Z 943.69,A -85,B 0,C 180,E1 21630.521,E2 21630.521} C_VEL
LIN {X 0,Y 396.08,Z 949.237,A -85,B 0,C 180,E1 21631.451,E2 21631.451} C_VEL
LIN {X 0,Y 379.297,Z 988.682,A -85,B 0,C 180,E1 21634.929,E2 21634.929} C_VEL
LIN {X 0,Y 361.122,Z 1024.334,A -85,B 0,C 180,E1 21639.416,E2 21639.416} C_VEL
LIN {X 0,Y 343.403,Z 1054.878,A -85,B 0,C 180,E1 21644.861,E2 21644.861} C_VEL
LIN {X 0,Y 328.34,Z 1079.517,A -85,B 0,C 180,E1 21651.111,E2 21651.111} C_VEL
LIN {X 0,Y 316.103,Z 1099.463,A -85,B 0,C 180,E1 21658.277,E2 21658.277} C_VEL
LIN {X 0,Y 307.327,Z 1115.226,A -85,B 0,C 180,E1 21666.838,E2 21666.838} C_VEL
LIN {X 0,Y 303.491,Z 1123.541,A -85,B 0,C 180,E1 21674.108,E2 21674.108} C_VEL
LIN {X 0,Y 301.826,Z 1127.89,A -85,B 0,C 180,E1 21681.363,E2 21681.363} C_VEL
LIN {X 0,Y 301.742,Z 1128.679,A -85,B 0,C 180,E1 21687.131,E2 21687.131} C_VEL
LIN {X 0,Y 302.166,Z 1127.129,A -85,B 0,C 180,E1 21692.868,E2 21692.868} C_VEL
LIN {X 0,Y 303.505,Z 1121.711,A -85,B 0,C 180,E1 21700.037,E2 21700.037} C_VEL
LIN {X 0,Y 307.621,Z 1111.298,A -85,B 0,C 180,E1 21707.881,E2 21707.881} C_VEL
LIN {X 0,Y 315.36,Z 1095.546,A -85,B 0,C 180,E1 21715.549,E2 21715.549} C_VEL
LIN {X 0,Y 327.309,Z 1073.802,A -85,B 0,C 180,E1 21722.854,E2 21722.854} C_VEL
LIN {X 0,Y 341.911,Z 1047.557,A -85,B 0,C 180,E1 21729.064,E2 21729.064} C_VEL
LIN {X 0,Y 359.416,Z 1013.703,A -85,B 0,C 180,E1 21734.69,E2 21734.69} C_VEL
LIN {X 0,Y 376.583,Z 975.892,A -85,B 0,C 180,E1 21739.063,E2 21739.063} C_VEL
LIN {X 0,Y 389.081,Z 942.899,A -85,B 0,C 180,E1 21741.847,E2 21741.847} C_VEL
LIN {X 0,Y 384.236,Z 917.016,A -85,B 0,C 180,E1 21746.595,E2 21746.595} C_VEL
LIN {X 0,Y 376.408,Z 891.922,A -85,B 0,C 180,E1 21752.148,E2 21752.148} C_VEL
LIN {X 0,Y 368.12,Z 872.13,A -85,B 0,C 180,E1 21757.923,E2 21757.923} C_VEL
LIN {X 0,Y 361.55,Z 859.105,A -85,B 0,C 180,E1 21763.226,E2 21763.226} C_VEL
LIN {X 0,Y 356.827,Z 849.496,A -85,B 0,C 180,E1 21768.532,E2 21768.532} C_VEL
LIN {X 0,Y 353.94,Z 842.901,A -85,B 0,C 180,E1 21775.099,E2 21775.099} C_VEL
LIN {X 0,Y 354.501,Z 843.743,A -85,B 0,C 180,E1 21782.821,E2 21782.821} C_VEL
LIN {X 0,Y 358.224,Z 851.357,A -85,B 0,C 180,E1 21789.096,E2 21789.096} C_VEL
LIN {X 0,Y 362.761,Z 859.767,A -85,B 0,C 180,E1 21793.545,E2 21793.545} C_VEL
LIN {X 0,Y 370.058,Z 873.292,A -85,B 0,C 180,E1 21798.828,E2 21798.828} C_VEL
LIN {X 0,Y 378.926,Z 893.027,A -85,B 0,C 180,E1 21804.287,E2 21804.287} C_VEL
LIN {X 0,Y 387.249,Z 916.495,A -85,B 0,C 180,E1 21809.249,E2 21809.249} C_VEL
LIN {X 0,Y 393.034,Z 940.284,A -85,B 0,C 180,E1 21813.42,E2 21813.42} C_VEL
LIN {X 0,Y 379.579,Z 979.4,A -85,B 0,C 180,E1 21816.276,E2 21816.276} C_VEL
LIN {X 0,Y 363.015,Z 1017.962,A -85,B 0,C 180,E1 21820.145,E2 21820.145} C_VEL
LIN {X 0,Y 345.587,Z 1053.42,A -85,B 0,C 180,E1 21825.237,E2 21825.237} C_VEL
LIN {X 0,Y 330.194,Z 1082.534,A -85,B 0,C 180,E1 21831.155,E2 21831.155} C_VEL
LIN {X 0,Y 318,Z 1105.666,A -85,B 0,C 180,E1 21837.682,E2 21837.682} C_VEL
LIN {X 0,Y 308.695,Z 1125.405,A -85,B 0,C 180,E1 21845.561,E2 21845.561} C_VEL
LIN {X 0,Y 303.499,Z 1139.539,A -85,B 0,C 180,E1 21854.105,E2 21854.105} C_VEL
LIN {X 0,Y 301.993,Z 1146.871,A -85,B 0,C 180,E1 21861.365,E2 21861.365} C_VEL
LIN {X 0,Y 301.878,Z 1149.732,A -85,B 0,C 180,E1 21867.129,E2 21867.129} C_VEL
LIN {X 0,Y 301.815,Z 1149.991,A -85,B 0,C 180,E1 21872.868,E2 21872.868} C_VEL
LIN {X 0,Y 302.166,Z 1146.834,A -85,B 0,C 180,E1 21880.079,E2 21880.079} C_VEL
LIN {X 0,Y 304.167,Z 1139.591,A -85,B 0,C 180,E1 21887.341,E2 21887.341} C_VEL
LIN {X 0,Y 310.443,Z 1125.401,A -85,B 0,C 180,E1 21895.98,E2 21895.98} C_VEL
LIN {X 0,Y 321.858,Z 1104.404,A -85,B 0,C 180,E1 21904.289,E2 21904.289} C_VEL
LIN {X 0,Y 337.399,Z 1078.128,A -85,B 0,C 180,E1 21911.344,E2 21911.344} C_VEL
LIN {X 0,Y 354.42,Z 1048.13,A -85,B 0,C 180,E1 21917,E2 21917} C_VEL
LIN {X 0,Y 371.856,Z 1014.788,A -85,B 0,C 180,E1 21921.466,E2 21921.466} C_VEL
LIN {X 0,Y 389.698,Z 975.539,A -85,B 0,C 180,E1 21925.151,E2 21925.151} C_VEL
LIN {X 0,Y 400.631,Z 945.66,A -85,B 0,C 180,E1 21927.288,E2 21927.288} C_VEL
LIN {X 0,Y 394.699,Z 921.832,A -85,B 0,C 180,E1 21932.04,E2 21932.04} C_VEL
LIN {X 0,Y 387.738,Z 901.821,A -85,B 0,C 180,E1 21937.071,E2 21937.071} C_VEL
LIN {X 0,Y 381.327,Z 887.109,A -85,B 0,C 180,E1 21941.997,E2 21941.997} C_VEL
LIN {X 0,Y 376.346,Z 876.718,A -85,B 0,C 180,E1 21946.802,E2 21946.802} C_VEL
LIN {X 0,Y 373.713,Z 871.28,A -85,B 0,C 180,E1 21950.257,E2 21950.257} C_VEL
LIN {X 0,Y 372.386,Z 868.772,A -85,B 0,C 180,E1 21952.606,E2 21952.606} C_VEL
LIN {X 0,Y 371.038,Z 869.108,A -85,B 0,C 180,E1 21954.617,E2 21954.617} C_VEL
LIN {X 0,Y 368.874,Z 872.931,A -85,B 0,C 180,E1 21958.007,E2 21958.007} C_VEL
LIN {X 0,Y 369.571,Z 874.303,A -85,B 0,C 180,E1 21963.593,E2 21963.593} C_VEL
LIN {X 0,Y 371.697,Z 880.548,A -85,B 0,C 180,E1 21968.771,E2 21968.771} C_VEL
LIN {X 0,Y 376.139,Z 891.934,A -85,B 0,C 180,E1 21974.602,E2 21974.602} C_VEL
LIN {X 0,Y 382.321,Z 909.794,A -85,B 0,C 180,E1 21980.838,E2 21980.838} C_VEL
LIN {X 0,Y 387.826,Z 931.29,A -85,B 0,C 180,E1 21986.345,E2 21986.345} C_VEL
LIN {X 0,Y 390.713,Z 952.114,A -85,B 0,C 180,E1 21990.667,E2 21990.667} C_VEL
LIN {X 0,Y 374.106,Z 989.891,A -85,B 0,C 180,E1 21994.042,E2 21994.042} C_VEL
LIN {X 0,Y 355.588,Z 1025.144,A -85,B 0,C 180,E1 21998.512,E2 21998.512} C_VEL
LIN {X 0,Y 336.901,Z 1056.249,A -85,B 0,C 180,E1 22004.141,E2 22004.141} C_VEL
LIN {X 0,Y 321.327,Z 1080.688,A -85,B 0,C 180,E1 22010.509,E2 22010.509} C_VEL
LIN {X 0,Y 309.137,Z 1099.658,A -85,B 0,C 180,E1 22017.475,E2 22017.475} C_VEL
LIN {X 0,Y 299.857,Z 1115.444,A -85,B 0,C 180,E1 22026.226,E2 22026.226} C_VEL
LIN {X 0,Y 295.265,Z 1124.957,A -85,B 0,C 180,E1 22035.175,E2 22035.175} C_VEL
LIN {X 0,Y 293.814,Z 1128.855,A -85,B 0,C 180,E1 22044.098,E2 22044.098} C_VEL
LIN {X 0,Y 294.125,Z 1128.488,A -85,B 0,C 180,E1 22050.002,E2 22050.002} C_VEL
LIN {X 0,Y 294.921,Z 1124.623,A -85,B 0,C 180,E1 22057.361,E2 22057.361} C_VEL
LIN {X 0,Y 298.284,Z 1115.617,A -85,B 0,C 180,E1 22065.751,E2 22065.751} C_VEL
LIN {X 0,Y 306.379,Z 1099.302,A -85,B 0,C 180,E1 22074.788,E2 22074.788} C_VEL
LIN {X 0,Y 319.31,Z 1076.567,A -85,B 0,C 180,E1 22082.974,E2 22082.974} C_VEL
LIN {X 0,Y 335.031,Z 1049.243,A -85,B 0,C 180,E1 22089.668,E2 22089.668} C_VEL
LIN {X 0,Y 352.337,Z 1016.993,A -85,B 0,C 180,E1 22095.194,E2 22095.194} C_VEL
LIN {X 0,Y 368.601,Z 982.872,A -85,B 0,C 180,E1 22099.34,E2 22099.34} C_VEL
LIN {X 0,Y 383.377,Z 945.116,A -85,B 0,C 180,E1 22102.74,E2 22102.74} C_VEL
LIN {X 0,Y 378.731,Z 919.466,A -85,B 0,C 180,E1 22107.665,E2 22107.665} C_VEL
LIN {X 0,Y 371.295,Z 894.989,A -85,B 0,C 180,E1 22113.406,E2 22113.406} C_VEL
LIN {X 0,Y 364.352,Z 877.807,A -85,B 0,C 180,E1 22118.722,E2 22118.722} C_VEL
LIN {X 0,Y 358.334,Z 864.899,A -85,B 0,C 180,E1 22124.169,E2 22124.169} C_VEL
LIN {X 0,Y 354.262,Z 856.56,A -85,B 0,C 180,E1 22129.397,E2 22129.397} C_VEL
LIN {X 0,Y 352.175,Z 850.605,A -85,B 0,C 180,E1 22135.074,E2 22135.074} C_VEL
LIN {X 0,Y 352.676,Z 851.398,A -85,B 0,C 180,E1 22142.624,E2 22142.624} C_VEL
LIN {X 0,Y 356.207,Z 859.11,A -85,B 0,C 180,E1 22148.995,E2 22148.995} C_VEL
LIN {X 0,Y 360.273,Z 866.936,A -85,B 0,C 180,E1 22153.197,E2 22153.197} C_VEL
LIN {X 0,Y 367.106,Z 880.431,A -85,B 0,C 180,E1 22158.518,E2 22158.518} C_VEL
LIN {X 0,Y 375.429,Z 900.113,A -85,B 0,C 180,E1 22164.042,E2 22164.042} C_VEL
LIN {X 0,Y 382.692,Z 922.702,A -85,B 0,C 180,E1 22168.919,E2 22168.919} C_VEL
LIN {X 0,Y 387.516,Z 943.961,A -85,B 0,C 180,E1 22172.746,E2 22172.746} C_VEL
LIN {X 0,Y 372.489,Z 984.464,A -85,B 0,C 180,E1 22175.769,E2 22175.769} C_VEL
LIN {X 0,Y 356.622,Z 1019.891,A -85,B 0,C 180,E1 22179.451,E2 22179.451} C_VEL
LIN {X 0,Y 339.071,Z 1054.422,A -85,B 0,C 180,E1 22184.514,E2 22184.514} C_VEL
LIN {X 0,Y 321.798,Z 1085.91,A -85,B 0,C 180,E1 22191.168,E2 22191.168} C_VEL
LIN {X 0,Y 308.205,Z 1110.844,A -85,B 0,C 180,E1 22198.84,E2 22198.84} C_VEL
LIN {X 0,Y 299.498,Z 1128.912,A -85,B 0,C 180,E1 22206.98,E2 22206.98} C_VEL
LIN {X 0,Y 295.228,Z 1141.003,A -85,B 0,C 180,E1 22215.17,E2 22215.17} C_VEL
LIN {X 0,Y 294.106,Z 1146.567,A -85,B 0,C 180,E1 22221.131,E2 22221.131} C_VEL
LIN {X 0,Y 293.967,Z 1149.438,A -85,B 0,C 180,E1 22227.052,E2 22227.052} C_VEL
LIN {X 0,Y 293.906,Z 1149.713,A -85,B 0,C 180,E1 22232.945,E2 22232.945} C_VEL
LIN {X 0,Y 294.295,Z 1146.57,A -85,B 0,C 180,E1 22240.351,E2 22240.351} C_VEL
LIN {X 0,Y 297.128,Z 1137.626,A -85,B 0,C 180,E1 22249.105,E2 22249.105} C_VEL
LIN {X 0,Y 303.863,Z 1123.659,A -85,B 0,C 180,E1 22257.385,E2 22257.385} C_VEL
LIN {X 0,Y 316.157,Z 1102.539,A -85,B 0,C 180,E1 22265.677,E2 22265.677} C_VEL
LIN {X 0,Y 332.935,Z 1075.268,A -85,B 0,C 180,E1 22272.905,E2 22272.905} C_VEL
LIN {X 0,Y 351.792,Z 1043.157,A -85,B 0,C 180,E1 22278.736,E2 22278.736} C_VEL
LIN {X 0,Y 370.937,Z 1006.678,A -85,B 0,C 180,E1 22283.321,E2 22283.321} C_VEL
LIN {X 0,Y 388.405,Z 967.572,A -85,B 0,C 180,E1 22286.729,E2 22286.729} C_VEL
LIN {X 0,Y 395.195,Z 949.052,A -85,B 0,C 180,E1 22288.058,E2 22288.058} C_VEL
LIN {X 0,Y 389.741,Z 925.721,A -85,B 0,C 180,E1 22292.907,E2 22292.907} C_VEL
LIN {X 0,Y 383.293,Z 906.376,A -85,B 0,C 180,E1 22298.012,E2 22298.012} C_VEL
LIN {X 0,Y 376.816,Z 890.495,A -85,B 0,C 180,E1 22303.704,E2 22303.704} C_VEL
LIN {X 0,Y 371.909,Z 879.348,A -85,B 0,C 180,E1 22309.729,E2 22309.729} C_VEL
LIN {X 0,Y 369.494,Z 873.332,A -85,B 0,C 180,E1 22315.313,E2 22315.313} C_VEL
LIN {X 0,Y 368.874,Z 872.931,A -85,B 0,C 180,E1 22318.007,E2 22318.007} C_VEL
LIN {X 0,Y 367.888,Z 876.625,A -85,B 0,C 180,E1 22320.654,E2 22320.654} C_VEL
LIN {X 0,Y 367.068,Z 881.627,A -85,B 0,C 180,E1 22323.3,E2 22323.3} C_VEL
LIN {X 0,Y 369.402,Z 889.386,A -85,B 0,C 180,E1 22329.419,E2 22329.419} C_VEL
LIN {X 0,Y 373.918,Z 901.823,A -85,B 0,C 180,E1 22335.56,E2 22335.56} C_VEL
LIN {X 0,Y 379.354,Z 919.808,A -85,B 0,C 180,E1 22341.519,E2 22341.519} C_VEL
LIN {X 0,Y 383.841,Z 941.693,A -85,B 0,C 180,E1 22347.026,E2 22347.026} C_VEL
LIN {X 0,Y 385.345,Z 955.16,A -85,B 0,C 180,E1 22349.872,E2 22349.872} C_VEL
LIN {X 0,Y 368.617,Z 991.833,A -85,B 0,C 180,E1 22353.211,E2 22353.211} C_VEL
LIN {X 0,Y 350.085,Z 1026.052,A -85,B 0,C 180,E1 22357.593,E2 22357.593} C_VEL
LIN {X 0,Y 330.346,Z 1057.796,A -85,B 0,C 180,E1 22363.432,E2 22363.432} C_VEL
LIN {X 0,Y 313.425,Z 1083.165,A -85,B 0,C 180,E1 22370.286,E2 22370.286} C_VEL
LIN {X 0,Y 300.248,Z 1102.838,A -85,B 0,C 180,E1 22378.084,E2 22378.084} C_VEL
LIN {X 0,Y 292.418,Z 1115.662,A -85,B 0,C 180,E1 22385.583,E2 22385.583} C_VEL
LIN {X 0,Y 288.013,Z 1124.039,A -85,B 0,C 180,E1 22393.23,E2 22393.23} C_VEL
LIN {X 0,Y 286.073,Z 1128.425,A -85,B 0,C 180,E1 22400.884,E2 22400.884} C_VEL
LIN {X 0,Y 285.948,Z 1129.252,A -85,B 0,C 180,E1 22406.973,E2 22406.973} C_VEL
LIN {X 0,Y 286.383,Z 1127.744,A -85,B 0,C 180,E1 22413.026,E2 22413.026} C_VEL
LIN {X 0,Y 287.894,Z 1122.372,A -85,B 0,C 180,E1 22420.588,E2 22420.588} C_VEL
LIN {X 0,Y 292.466,Z 1112.007,A -85,B 0,C 180,E1 22428.842,E2 22428.842} C_VEL
LIN {X 0,Y 300.982,Z 1096.329,A -85,B 0,C 180,E1 22436.864,E2 22436.864} C_VEL
LIN {X 0,Y 313.29,Z 1075.839,A -85,B 0,C 180,E1 22444.107,E2 22444.107} C_VEL
LIN {X 0,Y 329.982,Z 1047.945,A -85,B 0,C 180,E1 22450.925,E2 22450.925} C_VEL
LIN {X 0,Y 348.636,Z 1014.102,A -85,B 0,C 180,E1 22456.619,E2 22456.619} C_VEL
LIN {X 0,Y 366.87,Z 976.078,A -85,B 0,C 180,E1 22461.029,E2 22461.029} C_VEL
LIN {X 0,Y 377.801,Z 948.949,A -85,B 0,C 180,E1 22463.379,E2 22463.379} C_VEL
LIN {X 0,Y 373.73,Z 924.169,A -85,B 0,C 180,E1 22468.291,E2 22468.291} C_VEL
LIN {X 0,Y 367.399,Z 901.277,A -85,B 0,C 180,E1 22473.831,E2 22473.831} C_VEL
LIN {X 0,Y 361.031,Z 884.351,A -85,B 0,C 180,E1 22479.18,E2 22479.18} C_VEL
LIN {X 0,Y 354.869,Z 870.084,A -85,B 0,C 180,E1 22485.511,E2 22485.511} C_VEL
LIN {X 0,Y 351.926,Z 863.884,A -85,B 0,C 180,E1 22489.796,E2 22489.796} C_VEL
LIN {X 0,Y 350.338,Z 858.291,A -85,B 0,C 180,E1 22495.048,E2 22495.048} C_VEL
LIN {X 0,Y 350.759,Z 859.047,A -85,B 0,C 180,E1 22502.465,E2 22502.465} C_VEL
LIN {X 0,Y 354.006,Z 866.704,A -85,B 0,C 180,E1 22508.819,E2 22508.819} C_VEL
LIN {X 0,Y 359.073,Z 876.59,A -85,B 0,C 180,E1 22514.153,E2 22514.153} C_VEL
LIN {X 0,Y 366.578,Z 893.758,A -85,B 0,C 180,E1 22520.189,E2 22520.189} C_VEL
LIN {X 0,Y 374.506,Z 915.413,A -85,B 0,C 180,E1 22525.762,E2 22525.762} C_VEL
LIN {X 0,Y 380.656,Z 940.289,A -85,B 0,C 180,E1 22530.752,E2 22530.752} C_VEL
LIN {X 0,Y 381.553,Z 948.469,A -85,B 0,C 180,E1 22532.066,E2 22532.066} C_VEL
LIN {X 0,Y 364.721,Z 991.101,A -85,B 0,C 180,E1 22535.377,E2 22535.377} C_VEL
LIN {X 0,Y 346.434,Z 1029.597,A -85,B 0,C 180,E1 22539.753,E2 22539.753} C_VEL
LIN {X 0,Y 328.638,Z 1062.459,A -85,B 0,C 180,E1 22545.104,E2 22545.104} C_VEL
LIN {X 0,Y 313.384,Z 1088.966,A -85,B 0,C 180,E1 22551.18,E2 22551.18} C_VEL
LIN {X 0,Y 300.581,Z 1111.629,A -85,B 0,C 180,E1 22558.48,E2 22558.48} C_VEL
LIN {X 0,Y 291.434,Z 1129.931,A -85,B 0,C 180,E1 22567.113,E2 22567.113} C_VEL
LIN {X 0,Y 287.436,Z 1140.678,A -85,B 0,C 180,E1 22574.758,E2 22574.758} C_VEL
LIN {X 0,Y 286.229,Z 1146.262,A -85,B 0,C 180,E1 22580.885,E2 22580.885} C_VEL
LIN {X 0,Y 286.071,Z 1149.144,A -85,B 0,C 180,E1 22586.97,E2 22586.97} C_VEL
LIN {X 0,Y 286,Z 1149.435,A -85,B 0,C 180,E1 22593.027,E2 22593.027} C_VEL
LIN {X 0,Y 286.447,Z 1146.307,A -85,B 0,C 180,E1 22600.638,E2 22600.638} C_VEL
LIN {X 0,Y 289.302,Z 1137.855,A -85,B 0,C 180,E1 22609.266,E2 22609.266} C_VEL
LIN {X 0,Y 296.641,Z 1123.446,A -85,B 0,C 180,E1 22618.11,E2 22618.11} C_VEL
LIN {X 0,Y 309.568,Z 1102.358,A -85,B 0,C 180,E1 22626.557,E2 22626.557} C_VEL
LIN {X 0,Y 326.977,Z 1075.124,A -85,B 0,C 180,E1 22633.883,E2 22633.883} C_VEL
LIN {X 0,Y 346.484,Z 1043.047,A -85,B 0,C 180,E1 22639.746,E2 22639.746} C_VEL
LIN {X 0,Y 366.167,Z 1006.628,A -85,B 0,C 180,E1 22644.335,E2 22644.335} C_VEL
LIN {X 0,Y 383.618,Z 968.718,A -85,B 0,C 180,E1 22647.642,E2 22647.642} C_VEL
LIN {X 0,Y 389.766,Z 952.473,A -85,B 0,C 180,E1 22648.828,E2 22648.828} C_VEL
LIN {X 0,Y 385.007,Z 930.276,A -85,B 0,C 180,E1 22653.655,E2 22653.655} C_VEL
LIN {X 0,Y 378.933,Z 910.986,A -85,B 0,C 180,E1 22658.975,E2 22658.975} C_VEL
LIN {X 0,Y 372.996,Z 895.78,A -85,B 0,C 180,E1 22664.832,E2 22664.832} C_VEL
LIN {X 0,Y 368.749,Z 886.142,A -85,B 0,C 180,E1 22670.571,E2 22670.571} C_VEL
LIN {X 0,Y 367.214,Z 880.882,A -85,B 0,C 180,E1 22675.284,E2 22675.284} C_VEL
LIN {X 0,Y 366.971,Z 880.777,A -85,B 0,C 180,E1 22682.363,E2 22682.363} C_VEL
LIN {X 0,Y 367.068,Z 881.627,A -85,B 0,C 180,E1 22683.3,E2 22683.3} C_VEL
LIN {X 0,Y 366.443,Z 885.438,A -85,B 0,C 180,E1 22684.544,E2 22684.544} C_VEL
LIN {X 0,Y 365.213,Z 892.618,A -85,B 0,C 180,E1 22686.314,E2 22686.314} C_VEL
LIN {X 0,Y 365.272,Z 892.927,A -85,B 0,C 180,E1 22686.54,E2 22686.54} C_VEL
LIN {X 0,Y 368.468,Z 902.548,A -85,B 0,C 180,E1 22692.552,E2 22692.552} C_VEL
LIN {X 0,Y 372.801,Z 916.943,A -85,B 0,C 180,E1 22698.309,E2 22698.309} C_VEL
LIN {X 0,Y 376.996,Z 935.112,A -85,B 0,C 180,E1 22703.629,E2 22703.629} C_VEL
LIN {X 0,Y 379.885,Z 956.851,A -85,B 0,C 180,E1 22708.752,E2 22708.752} C_VEL
LIN {X 0,Y 378.299,Z 962.473,A -85,B 0,C 180,E1 22709.396,E2 22709.396} C_VEL
LIN {X 0,Y 359.742,Z 1000.398,A -85,B 0,C 180,E1 22713.096,E2 22713.096} C_VEL
LIN {X 0,Y 340.209,Z 1034.116,A -85,B 0,C 180,E1 22717.808,E2 22717.808} C_VEL
LIN {X 0,Y 321.559,Z 1062.613,A -85,B 0,C 180,E1 22723.493,E2 22723.493} C_VEL
LIN {X 0,Y 305.656,Z 1085.496,A -85,B 0,C 180,E1 22730.009,E2 22730.009} C_VEL
LIN {X 0,Y 291.315,Z 1106.077,A -85,B 0,C 180,E1 22738.756,E2 22738.756} C_VEL
LIN {X 0,Y 282.744,Z 1119.728,A -85,B 0,C 180,E1 22748.033,E2 22748.033} C_VEL
LIN {X 0,Y 279.722,Z 1125.455,A -85,B 0,C 180,E1 22754.331,E2 22754.331} C_VEL
LIN {X 0,Y 278.016,Z 1129.41,A -85,B 0,C 180,E1 22763.761,E2 22763.761} C_VEL
LIN {X 0,Y 278.343,Z 1129.081,A -85,B 0,C 180,E1 22770.002,E2 22770.002} C_VEL
LIN {X 0,Y 279.214,Z 1125.261,A -85,B 0,C 180,E1 22777.778,E2 22777.778} C_VEL
LIN {X 0,Y 283.287,Z 1115.695,A -85,B 0,C 180,E1 22787.061,E2 22787.061} C_VEL
LIN {X 0,Y 291.903,Z 1100.065,A -85,B 0,C 180,E1 22796.107,E2 22796.107} C_VEL
LIN {X 0,Y 305.987,Z 1077.408,A -85,B 0,C 180,E1 22804.607,E2 22804.607} C_VEL
LIN {X 0,Y 323.255,Z 1049.616,A -85,B 0,C 180,E1 22811.592,E2 22811.592} C_VEL
LIN {X 0,Y 340.991,Z 1018.656,A -85,B 0,C 180,E1 22816.989,E2 22816.989} C_VEL
LIN {X 0,Y 357.881,Z 985.347,A -85,B 0,C 180,E1 22821.125,E2 22821.125} C_VEL
LIN {X 0,Y 372.035,Z 951.242,A -85,B 0,C 180,E1 22824.328,E2 22824.328} C_VEL
LIN {X 0,Y 368.556,Z 927.8,A -85,B 0,C 180,E1 22829.172,E2 22829.172} C_VEL
LIN {X 0,Y 362.91,Z 905.815,A -85,B 0,C 180,E1 22834.736,E2 22834.736} C_VEL
LIN {X 0,Y 356.687,Z 888.137,A -85,B 0,C 180,E1 22840.67,E2 22840.67} C_VEL
LIN {X 0,Y 351.793,Z 876.657,A -85,B 0,C 180,E1 22846.333,E2 22846.333} C_VEL
LIN {X 0,Y 349.546,Z 871.344,A -85,B 0,C 180,E1 22850.04,E2 22850.04} C_VEL
LIN {X 0,Y 348.273,Z 865.922,A -85,B 0,C 180,E1 22855.019,E2 22855.019} C_VEL
LIN {X 0,Y 348.656,Z 866.55,A -85,B 0,C 180,E1 22862.247,E2 22862.247} C_VEL
LIN {X 0,Y 351.522,Z 873.97,A -85,B 0,C 180,E1 22868.516,E2 22868.516} C_VEL
LIN {X 0,Y 356.135,Z 883.445,A -85,B 0,C 180,E1 22873.724,E2 22873.724} C_VEL
LIN {X 0,Y 362.675,Z 899.242,A -85,B 0,C 180,E1 22879.463,E2 22879.463} C_VEL
LIN {X 0,Y 370.145,Z 921.504,A -85,B 0,C 180,E1 22885.375,E2 22885.375} C_VEL
LIN {X 0,Y 375.793,Z 946.649,A -85,B 0,C 180,E1 22890.498,E2 22890.498} C_VEL
LIN {X 0,Y 376.11,Z 951.088,A -85,B 0,C 180,E1 22891.245,E2 22891.245} C_VEL
LIN {X 0,Y 359.357,Z 992.1,A -85,B 0,C 180,E1 22894.476,E2 22894.476} C_VEL
LIN {X 0,Y 340.657,Z 1030.277,A -85,B 0,C 180,E1 22898.857,E2 22898.857} C_VEL
LIN {X 0,Y 322.149,Z 1063.304,A -85,B 0,C 180,E1 22904.327,E2 22904.327} C_VEL
LIN {X 0,Y 305.54,Z 1091.006,A -85,B 0,C 180,E1 22910.905,E2 22910.905} C_VEL
LIN {X 0,Y 293.043,Z 1112.2,A -85,B 0,C 180,E1 22918.038,E2 22918.038} C_VEL
LIN {X 0,Y 283.967,Z 1129.575,A -85,B 0,C 180,E1 22926.476,E2 22926.476} C_VEL
LIN {X 0,Y 279.689,Z 1140.353,A -85,B 0,C 180,E1 22934.326,E2 22934.326} C_VEL
LIN {X 0,Y 278.348,Z 1145.957,A -85,B 0,C 180,E1 22940.625,E2 22940.625} C_VEL
LIN {X 0,Y 278.159,Z 1148.85,A -85,B 0,C 180,E1 22946.884,E2 22946.884} C_VEL
LIN {X 0,Y 278.091,Z 1149.157,A -85,B 0,C 180,E1 22953.113,E2 22953.113} C_VEL
LIN {X 0,Y 278.602,Z 1146.044,A -85,B 0,C 180,E1 22960.941,E2 22960.941} C_VEL
LIN {X 0,Y 281.672,Z 1137.615,A -85,B 0,C 180,E1 22969.809,E2 22969.809} C_VEL
LIN {X 0,Y 289.468,Z 1123.232,A -85,B 0,C 180,E1 22978.871,E2 22978.871} C_VEL
LIN {X 0,Y 302.614,Z 1102.84,A -85,B 0,C 180,E1 22987.26,E2 22987.26} C_VEL
LIN {X 0,Y 321.157,Z 1074.979,A -85,B 0,C 180,E1 22994.89,E2 22994.89} C_VEL
LIN {X 0,Y 341.328,Z 1042.941,A -85,B 0,C 180,E1 23000.78,E2 23000.78} C_VEL
LIN {X 0,Y 360.918,Z 1007.729,A -85,B 0,C 180,E1 23005.249,E2 23005.249} C_VEL
LIN {X 0,Y 378.67,Z 970.441,A -85,B 0,C 180,E1 23008.54,E2 23008.54} C_VEL
LIN {X 0,Y 384.384,Z 955.99,A -85,B 0,C 180,E1 23009.611,E2 23009.611} C_VEL
LIN {X 0,Y 380.04,Z 934.306,A -85,B 0,C 180,E1 23014.53,E2 23014.53} C_VEL
LIN {X 0,Y 374.44,Z 915.231,A -85,B 0,C 180,E1 23020.098,E2 23020.098} C_VEL
LIN {X 0,Y 368.86,Z 900.162,A -85,B 0,C 180,E1 23026.381,E2 23026.381} C_VEL
LIN {X 0,Y 365.69,Z 892.884,A -85,B 0,C 180,E1 23031.391,E2 23031.391} C_VEL
LIN {X 0,Y 364.649,Z 888.501,A -85,B 0,C 180,E1 23035.25,E2 23035.25} C_VEL
LIN {X 0,Y 364.426,Z 888.316,A -85,B 0,C 180,E1 23042.38,E2 23042.38} C_VEL
LIN {X 0,Y 365.272,Z 892.927,A -85,B 0,C 180,E1 23046.54,E2 23046.54} C_VEL
LIN {X 0,Y 365.258,Z 897.559,A -85,B 0,C 180,E1 23048.459,E2 23048.459} C_VEL
LIN {X 0,Y 364.727,Z 908.03,A -85,B 0,C 180,E1 23051.535,E2 23051.535} C_VEL
LIN {X 0,Y 368.437,Z 921.675,A -85,B 0,C 180,E1 23057.337,E2 23057.337} C_VEL
LIN {X 0,Y 372.057,Z 939.043,A -85,B 0,C 180,E1 23062.736,E2 23062.736} C_VEL
LIN {X 0,Y 374.434,Z 958.995,A -85,B 0,C 180,E1 23067.65,E2 23067.65} C_VEL
LIN {X 0,Y 374.602,Z 961.928,A -85,B 0,C 180,E1 23068.28,E2 23068.28} C_VEL
LIN {X 0,Y 355.378,Z 1000.407,A -85,B 0,C 180,E1 23072,E2 23072} C_VEL
LIN {X 0,Y 336.03,Z 1032.98,A -85,B 0,C 180,E1 23076.505,E2 23076.505} C_VEL
LIN {X 0,Y 316.796,Z 1061.556,A -85,B 0,C 180,E1 23082.12,E2 23082.12} C_VEL
LIN {X 0,Y 298.637,Z 1086.691,A -85,B 0,C 180,E1 23089.371,E2 23089.371} C_VEL
LIN {X 0,Y 284.341,Z 1106.273,A -85,B 0,C 180,E1 23097.899,E2 23097.899} C_VEL
LIN {X 0,Y 275.208,Z 1119.958,A -85,B 0,C 180,E1 23107.398,E2 23107.398} C_VEL
LIN {X 0,Y 271.964,Z 1125.705,A -85,B 0,C 180,E1 23113.872,E2 23113.872} C_VEL
LIN {X 0,Y 270.11,Z 1129.688,A -85,B 0,C 180,E1 23123.578,E2 23123.578} C_VEL
LIN {X 0,Y 270.458,Z 1129.377,A -85,B 0,C 180,E1 23130.002,E2 23130.002} C_VEL
LIN {X 0,Y 271.369,Z 1125.579,A -85,B 0,C 180,E1 23138.004,E2 23138.004} C_VEL
LIN {X 0,Y 274.635,Z 1117.997,A -85,B 0,C 180,E1 23145.971,E2 23145.971} C_VEL
LIN {X 0,Y 281.966,Z 1104.859,A -85,B 0,C 180,E1 23154.569,E2 23154.569} C_VEL
LIN {X 0,Y 294.627,Z 1085.221,A -85,B 0,C 180,E1 23163.023,E2 23163.023} C_VEL
LIN {X 0,Y 311.461,Z 1059.428,A -85,B 0,C 180,E1 23170.462,E2 23170.462} C_VEL
LIN {X 0,Y 330.415,Z 1028.332,A -85,B 0,C 180,E1 23176.575,E2 23176.575} C_VEL
LIN {X 0,Y 348.929,Z 994.145,A -85,B 0,C 180,E1 23181.219,E2 23181.219} C_VEL
LIN {X 0,Y 365.889,Z 956.88,A -85,B 0,C 180,E1 23184.821,E2 23184.821} C_VEL
LIN {X 0,Y 366.134,Z 950.102,A -85,B 0,C 180,E1 23186.003,E2 23186.003} C_VEL
LIN {X 0,Y 362.532,Z 927.324,A -85,B 0,C 180,E1 23191.086,E2 23191.086} C_VEL
LIN {X 0,Y 357.72,Z 908.159,A -85,B 0,C 180,E1 23196.34,E2 23196.34} C_VEL
LIN {X 0,Y 352.568,Z 893.079,A -85,B 0,C 180,E1 23201.889,E2 23201.889} C_VEL
LIN {X 0,Y 348.446,Z 882.497,A -85,B 0,C 180,E1 23207.475,E2 23207.475} C_VEL
LIN {X 0,Y 346.065,Z 873.61,A -85,B 0,C 180,E1 23214.987,E2 23214.987} C_VEL
LIN {X 0,Y 346.404,Z 874.122,A -85,B 0,C 180,E1 23222.105,E2 23222.105} C_VEL
LIN {X 0,Y 348.978,Z 881.148,A -85,B 0,C 180,E1 23228.177,E2 23228.177} C_VEL
LIN {X 0,Y 353.278,Z 890.964,A -85,B 0,C 180,E1 23233.6,E2 23233.6} C_VEL
LIN {X 0,Y 359.598,Z 907.628,A -85,B 0,C 180,E1 23239.637,E2 23239.637} C_VEL
LIN {X 0,Y 366.032,Z 928.495,A -85,B 0,C 180,E1 23245.189,E2 23245.189} C_VEL
LIN {X 0,Y 370.727,Z 953.123,A -85,B 0,C 180,E1 23250.304,E2 23250.304} C_VEL
LIN {X 0,Y 354.298,Z 992.676,A -85,B 0,C 180,E1 23253.509,E2 23253.509} C_VEL
LIN {X 0,Y 335.611,Z 1029.692,A -85,B 0,C 180,E1 23257.754,E2 23257.754} C_VEL
LIN {X 0,Y 316.484,Z 1062.848,A -85,B 0,C 180,E1 23263.267,E2 23263.267} C_VEL
LIN {X 0,Y 299.218,Z 1090.59,A -85,B 0,C 180,E1 23269.915,E2 23269.915} C_VEL
LIN {X 0,Y 286.061,Z 1111.927,A -85,B 0,C 180,E1 23277.215,E2 23277.215} C_VEL
LIN {X 0,Y 276.496,Z 1129.217,A -85,B 0,C 180,E1 23285.8,E2 23285.8} C_VEL
LIN {X 0,Y 271.927,Z 1140.027,A -85,B 0,C 180,E1 23293.866,E2 23293.866} C_VEL
LIN {X 0,Y 270.493,Z 1145.651,A -85,B 0,C 180,E1 23300.35,E2 23300.35} C_VEL
LIN {X 0,Y 270.249,Z 1148.555,A -85,B 0,C 180,E1 23306.793,E2 23306.793} C_VEL
LIN {X 0,Y 270.191,Z 1148.88,A -85,B 0,C 180,E1 23313.204,E2 23313.204} C_VEL
LIN {X 0,Y 270.749,Z 1145.78,A -85,B 0,C 180,E1 23321.263,E2 23321.263} C_VEL
LIN {X 0,Y 274.063,Z 1137.316,A -85,B 0,C 180,E1 23330.432,E2 23330.432} C_VEL
LIN {X 0,Y 282.346,Z 1123.02,A -85,B 0,C 180,E1 23339.671,E2 23339.671} C_VEL
LIN {X 0,Y 296.89,Z 1101.585,A -85,B 0,C 180,E1 23348.57,E2 23348.57} C_VEL
LIN {X 0,Y 315.457,Z 1074.833,A -85,B 0,C 180,E1 23355.931,E2 23355.931} C_VEL
LIN {X 0,Y 336.26,Z 1042.833,A -85,B 0,C 180,E1 23361.85,E2 23361.85} C_VEL
LIN {X 0,Y 356.559,Z 1007.418,A -85,B 0,C 180,E1 23366.335,E2 23366.335} C_VEL
LIN {X 0,Y 374.821,Z 969.938,A -85,B 0,C 180,E1 23369.616,E2 23369.616} C_VEL
LIN {X 0,Y 379.024,Z 960.254,A -85,B 0,C 180,E1 23370.302,E2 23370.302} C_VEL
LIN {X 0,Y 375.48,Z 939.946,A -85,B 0,C 180,E1 23375.012,E2 23375.012} C_VEL
LIN {X 0,Y 370.538,Z 921.551,A -85,B 0,C 180,E1 23380.516,E2 23380.516} C_VEL
LIN {X 0,Y 365.519,Z 906.79,A -85,B 0,C 180,E1 23386.863,E2 23386.863} C_VEL
LIN {X 0,Y 362.355,Z 898.816,A -85,B 0,C 180,E1 23392.818,E2 23392.818} C_VEL
LIN {X 0,Y 362.021,Z 896.087,A -85,B 0,C 180,E1 23395.216,E2 23395.216} C_VEL
LIN {X 0,Y 361.744,Z 895.832,A -85,B 0,C 180,E1 23402.397,E2 23402.397} C_VEL
LIN {X 0,Y 363.657,Z 904.613,A -85,B 0,C 180,E1 23409.57,E2 23409.57} C_VEL
LIN {X 0,Y 364.727,Z 908.03,A -85,B 0,C 180,E1 23411.535,E2 23411.535} C_VEL
LIN {X 0,Y 364.682,Z 914.129,A -85,B 0,C 180,E1 23413.363,E2 23413.363} C_VEL
LIN {X 0,Y 363.976,Z 926.198,A -85,B 0,C 180,E1 23416.284,E2 23416.284} C_VEL
LIN {X 0,Y 367.136,Z 942.766,A -85,B 0,C 180,E1 23421.742,E2 23421.742} C_VEL
LIN {X 0,Y 369.15,Z 962.267,A -85,B 0,C 180,E1 23426.761,E2 23426.761} C_VEL
LIN {X 0,Y 368.744,Z 966.305,A -85,B 0,C 180,E1 23427.55,E2 23427.55} C_VEL
LIN {X 0,Y 349.249,Z 1003.854,A -85,B 0,C 180,E1 23431.277,E2 23431.277} C_VEL
LIN {X 0,Y 327.439,Z 1038.958,A -85,B 0,C 180,E1 23436.363,E2 23436.363} C_VEL
LIN {X 0,Y 306.348,Z 1068.632,A -85,B 0,C 180,E1 23442.739,E2 23442.739} C_VEL
LIN {X 0,Y 288.346,Z 1092.036,A -85,B 0,C 180,E1 23450.272,E2 23450.272} C_VEL
LIN {X 0,Y 274.863,Z 1109.826,A -85,B 0,C 180,E1 23459,E2 23459} C_VEL
LIN {X 0,Y 266.92,Z 1121.468,A -85,B 0,C 180,E1 23467.938,E2 23467.938} C_VEL
LIN {X 0,Y 262.938,Z 1128.36,A -85,B 0,C 180,E1 23477.664,E2 23477.664} C_VEL
LIN {X 0,Y 262.238,Z 1130.113,A -85,B 0,C 180,E1 23486.699,E2 23486.699} C_VEL
LIN {X 0,Y 262.735,Z 1128.661,A -85,B 0,C 180,E1 23493.299,E2 23493.299} C_VEL
LIN {X 0,Y 264.533,Z 1123.361,A -85,B 0,C 180,E1 23501.535,E2 23501.535} C_VEL
LIN {X 0,Y 270.632,Z 1111.933,A -85,B 0,C 180,E1 23511.282,E2 23511.282} C_VEL
LIN {X 0,Y 282.443,Z 1093.667,A -85,B 0,C 180,E1 23520.791,E2 23520.791} C_VEL
LIN {X 0,Y 299.355,Z 1068.917,A -85,B 0,C 180,E1 23529.125,E2 23529.125} C_VEL
LIN {X 0,Y 318.698,Z 1039.284,A -85,B 0,C 180,E1 23535.763,E2 23535.763} C_VEL
LIN {X 0,Y 338.275,Z 1005.539,A -85,B 0,C 180,E1 23540.953,E2 23540.953} C_VEL
LIN {X 0,Y 356.057,Z 969.831,A -85,B 0,C 180,E1 23544.776,E2 23544.776} C_VEL
LIN {X 0,Y 360.959,Z 957.938,A -85,B 0,C 180,E1 23545.88,E2 23545.88} C_VEL
LIN {X 0,Y 358.532,Z 936.288,A -85,B 0,C 180,E1 23550.732,E2 23550.732} C_VEL
LIN {X 0,Y 354.308,Z 916.584,A -85,B 0,C 180,E1 23556.099,E2 23556.099} C_VEL
LIN {X 0,Y 350.056,Z 902.116,A -85,B 0,C 180,E1 23561.24,E2 23561.24} C_VEL
LIN {X 0,Y 345.892,Z 890.235,A -85,B 0,C 180,E1 23567.381,E2 23567.381} C_VEL
LIN {X 0,Y 343.619,Z 881.394,A -85,B 0,C 180,E1 23574.951,E2 23574.951} C_VEL
LIN {X 0,Y 343.651,Z 880.801,A -85,B 0,C 180,E1 23579.996,E2 23579.996} C_VEL
LIN {X 0,Y 346.062,Z 887.6,A -85,B 0,C 180,E1 23587.522,E2 23587.522} C_VEL
LIN {X 0,Y 350.529,Z 899.04,A -85,B 0,C 180,E1 23593.709,E2 23593.709} C_VEL
LIN {X 0,Y 356.492,Z 915.872,A -85,B 0,C 180,E1 23599.815,E2 23599.815} C_VEL
LIN {X 0,Y 361.982,Z 936.773,A -85,B 0,C 180,E1 23605.325,E2 23605.325} C_VEL
LIN {X 0,Y 365.014,Z 957.5,A -85,B 0,C 180,E1 23609.612,E2 23609.612} C_VEL
LIN {X 0,Y 348.046,Z 995.795,A -85,B 0,C 180,E1 23612.755,E2 23612.755} C_VEL
LIN {X 0,Y 329.789,Z 1030.725,A -85,B 0,C 180,E1 23616.852,E2 23616.852} C_VEL
LIN {X 0,Y 309.953,Z 1064.019,A -85,B 0,C 180,E1 23622.489,E2 23622.489} C_VEL
LIN {X 0,Y 291.424,Z 1092.631,A -85,B 0,C 180,E1 23629.595,E2 23629.595} C_VEL
LIN {X 0,Y 276.857,Z 1115.277,A -85,B 0,C 180,E1 23637.933,E2 23637.933} C_VEL
LIN {X 0,Y 267.775,Z 1131.348,A -85,B 0,C 180,E1 23646.731,E2 23646.731} C_VEL
LIN {X 0,Y 263.609,Z 1141.319,A -85,B 0,C 180,E1 23655.049,E2 23655.049} C_VEL
LIN {X 0,Y 262.306,Z 1147.127,A -85,B 0,C 180,E1 23663.382,E2 23663.382} C_VEL
LIN {X 0,Y 262.56,Z 1148.759,A -85,B 0,C 180,E1 23669.998,E2 23669.998} C_VEL
LIN {X 0,Y 262.305,Z 1147.822,A -85,B 0,C 180,E1 23676.614,E2 23676.614} C_VEL
LIN {X 0,Y 263.661,Z 1143.124,A -85,B 0,C 180,E1 23684.944,E2 23684.944} C_VEL
LIN {X 0,Y 268.63,Z 1133.234,A -85,B 0,C 180,E1 23694.066,E2 23694.066} C_VEL
LIN {X 0,Y 279.705,Z 1116.485,A -85,B 0,C 180,E1 23703.623,E2 23703.623} C_VEL
LIN {X 0,Y 296.116,Z 1093.825,A -85,B 0,C 180,E1 23712.006,E2 23712.006} C_VEL
LIN {X 0,Y 316.937,Z 1064.444,A -85,B 0,C 180,E1 23719.189,E2 23719.189} C_VEL
LIN {X 0,Y 338.985,Z 1030.363,A -85,B 0,C 180,E1 23724.716,E2 23724.716} C_VEL
LIN {X 0,Y 359.216,Z 994.167,A -85,B 0,C 180,E1 23728.7,E2 23728.7} C_VEL
LIN {X 0,Y 373.373,Z 964.319,A -85,B 0,C 180,E1 23731.084,E2 23731.084} C_VEL
LIN {X 0,Y 371.532,Z 948.688,A -85,B 0,C 180,E1 23734.667,E2 23734.667} C_VEL
LIN {X 0,Y 367.133,Z 929.518,A -85,B 0,C 180,E1 23740.361,E2 23740.361} C_VEL
LIN {X 0,Y 362.628,Z 914.916,A -85,B 0,C 180,E1 23746.52,E2 23746.52} C_VEL
LIN {X 0,Y 359.915,Z 907.567,A -85,B 0,C 180,E1 23751.555,E2 23751.555} C_VEL
LIN {X 0,Y 359.12,Z 903.566,A -85,B 0,C 180,E1 23755.177,E2 23755.177} C_VEL
LIN {X 0,Y 358.839,Z 903.303,A -85,B 0,C 180,E1 23762.417,E2 23762.417} C_VEL
LIN {X 0,Y 360.061,Z 910.243,A -85,B 0,C 180,E1 23768.449,E2 23768.449} C_VEL
LIN {X 0,Y 363.017,Z 921.68,A -85,B 0,C 180,E1 23774.464,E2 23774.464} C_VEL
LIN {X 0,Y 363.976,Z 926.198,A -85,B 0,C 180,E1 23776.284,E2 23776.284} C_VEL
LIN {X 0,Y 363.84,Z 933.287,A -85,B 0,C 180,E1 23778.027,E2 23778.027} C_VEL
LIN {X 0,Y 362.309,Z 946.801,A -85,B 0,C 180,E1 23780.79,E2 23780.79} C_VEL
LIN {X 0,Y 363.853,Z 966.248,A -85,B 0,C 180,E1 23786.036,E2 23786.036} C_VEL
LIN {X 0,Y 362.923,Z 970.665,A -85,B 0,C 180,E1 23786.8,E2 23786.8} C_VEL
LIN {X 0,Y 344.022,Z 1005.66,A -85,B 0,C 180,E1 23790.343,E2 23790.343} C_VEL
LIN {X 0,Y 323.122,Z 1038.367,A -85,B 0,C 180,E1 23795.078,E2 23795.078} C_VEL
LIN {X 0,Y 301.683,Z 1067.607,A -85,B 0,C 180,E1 23801.296,E2 23801.296} C_VEL
LIN {X 0,Y 283.712,Z 1090.204,A -85,B 0,C 180,E1 23808.435,E2 23808.435} C_VEL
LIN {X 0,Y 269.404,Z 1108.142,A -85,B 0,C 180,E1 23816.925,E2 23816.925} C_VEL
LIN {X 0,Y 260.286,Z 1120.417,A -85,B 0,C 180,E1 23826.024,E2 23826.024} C_VEL
LIN {X 0,Y 256.52,Z 1126.204,A -85,B 0,C 180,E1 23832.872,E2 23832.872} C_VEL
LIN {X 0,Y 254.306,Z 1130.244,A -85,B 0,C 180,E1 23843.177,E2 23843.177} C_VEL
LIN {X 0,Y 254.665,Z 1129.97,A -85,B 0,C 180,E1 23850.002,E2 23850.002} C_VEL
LIN {X 0,Y 255.698,Z 1126.216,A -85,B 0,C 180,E1 23858.498,E2 23858.498} C_VEL
LIN {X 0,Y 259.359,Z 1118.68,A -85,B 0,C 180,E1 23866.939,E2 23866.939} C_VEL
LIN {X 0,Y 267.711,Z 1105.327,A -85,B 0,C 180,E1 23876.144,E2 23876.144} C_VEL
LIN {X 0,Y 281.327,Z 1086.052,A -85,B 0,C 180,E1 23884.802,E2 23884.802} C_VEL
LIN {X 0,Y 299.909,Z 1059.718,A -85,B 0,C 180,E1 23892.596,E2 23892.596} C_VEL
LIN {X 0,Y 320.736,Z 1027.666,A -85,B 0,C 180,E1 23898.925,E2 23898.925} C_VEL
LIN {X 0,Y 341.042,Z 991.865,A -85,B 0,C 180,E1 23903.696,E2 23903.696} C_VEL
LIN {X 0,Y 355.508,Z 961.568,A -85,B 0,C 180,E1 23906.641,E2 23906.641} C_VEL
LIN {X 0,Y 353.462,Z 940.202,A -85,B 0,C 180,E1 23911.602,E2 23911.602} C_VEL
LIN {X 0,Y 349.806,Z 920.973,A -85,B 0,C 180,E1 23917.121,E2 23917.121} C_VEL
LIN {X 0,Y 345.744,Z 906.26,A -85,B 0,C 180,E1 23922.787,E2 23922.787} C_VEL
LIN {X 0,Y 342.392,Z 895.424,A -85,B 0,C 180,E1 23928.891,E2 23928.891} C_VEL
LIN {X 0,Y 341.035,Z 889.065,A -85,B 0,C 180,E1 23934.913,E2 23934.913} C_VEL
LIN {X 0,Y 341.108,Z 888.321,A -85,B 0,C 180,E1 23939.996,E2 23939.996} C_VEL
LIN {X 0,Y 343.44,Z 895.419,A -85,B 0,C 180,E1 23947.58,E2 23947.58} C_VEL
LIN {X 0,Y 347.411,Z 906.572,A -85,B 0,C 180,E1 23953.669,E2 23953.669} C_VEL
LIN {X 0,Y 352.453,Z 922.15,A -85,B 0,C 180,E1 23959.395,E2 23959.395} C_VEL
LIN {X 0,Y 357.412,Z 943.03,A -85,B 0,C 180,E1 23965.002,E2 23965.002} C_VEL
LIN {X 0,Y 359.845,Z 959.878,A -85,B 0,C 180,E1 23968.686,E2 23968.686} C_VEL
LIN {X 0,Y 341.424,Z 999.826,A -85,B 0,C 180,E1 23972.07,E2 23972.07} C_VEL
LIN {X 0,Y 322.944,Z 1033.63,A -85,B 0,C 180,E1 23976.199,E2 23976.199} C_VEL
LIN {X 0,Y 303.457,Z 1065.094,A -85,B 0,C 180,E1 23981.671,E2 23981.671} C_VEL
LIN {X 0,Y 284.318,Z 1093.592,A -85,B 0,C 180,E1 23988.937,E2 23988.937} C_VEL
LIN {X 0,Y 268.99,Z 1116.428,A -85,B 0,C 180,E1 23997.7,E2 23997.7} C_VEL
LIN {X 0,Y 259.705,Z 1132.184,A -85,B 0,C 180,E1 24006.872,E2 24006.872} C_VEL
LIN {X 0,Y 255.348,Z 1142.537,A -85,B 0,C 180,E1 24016.305,E2 24016.305} C_VEL
LIN {X 0,Y 254.402,Z 1146.823,A -85,B 0,C 180,E1 24023.175,E2 24023.175} C_VEL
LIN {X 0,Y 254.665,Z 1148.473,A -85,B 0,C 180,E1 24029.998,E2 24029.998} C_VEL
LIN {X 0,Y 254.403,Z 1147.552,A -85,B 0,C 180,E1 24036.821,E2 24036.821} C_VEL
LIN {X 0,Y 255.885,Z 1142.867,A -85,B 0,C 180,E1 24045.409,E2 24045.409} C_VEL
LIN {X 0,Y 261.203,Z 1133.002,A -85,B 0,C 180,E1 24054.796,E2 24054.796} C_VEL
LIN {X 0,Y 272.908,Z 1116.282,A -85,B 0,C 180,E1 24064.577,E2 24064.577} C_VEL
LIN {X 0,Y 290.664,Z 1092.906,A -85,B 0,C 180,E1 24073.312,E2 24073.312} C_VEL
LIN {X 0,Y 311.653,Z 1064.305,A -85,B 0,C 180,E1 24080.327,E2 24080.327} C_VEL
LIN {X 0,Y 334.664,Z 1029.85,A -85,B 0,C 180,E1 24085.903,E2 24085.903} C_VEL
LIN {X 0,Y 355.78,Z 992.881,A -85,B 0,C 180,E1 24089.924,E2 24089.924} C_VEL
LIN {X 0,Y 368.371,Z 966.292,A -85,B 0,C 180,E1 24092.126,E2 24092.126} C_VEL
LIN {X 0,Y 365.223,Z 945.564,A -85,B 0,C 180,E1 24097.59,E2 24097.59} C_VEL
LIN {X 0,Y 361.476,Z 930.023,A -85,B 0,C 180,E1 24102.992,E2 24102.992} C_VEL
LIN {X 0,Y 358.531,Z 919.978,A -85,B 0,C 180,E1 24107.84,E2 24107.84} C_VEL
LIN {X 0,Y 356.187,Z 911.039,A -85,B 0,C 180,E1 24115.137,E2 24115.137} C_VEL
LIN {X 0,Y 355.676,Z 910.016,A -85,B 0,C 180,E1 24120.004,E2 24120.004} C_VEL
LIN {X 0,Y 355.754,Z 912.033,A -85,B 0,C 180,E1 24123.656,E2 24123.656} C_VEL
LIN {X 0,Y 357.252,Z 919.604,A -85,B 0,C 180,E1 24129.743,E2 24129.743} C_VEL
LIN {X 0,Y 359.855,Z 932.085,A -85,B 0,C 180,E1 24135.716,E2 24135.716} C_VEL
LIN {X 0,Y 362.309,Z 946.801,A -85,B 0,C 180,E1 24140.79,E2 24140.79} C_VEL
LIN {X 0,Y 361.457,Z 954.754,A -85,B 0,C 180,E1 24142.438,E2 24142.438} C_VEL
LIN {X 0,Y 358.555,Z 969.327,A -85,B 0,C 180,E1 24145.058,E2 24145.058} C_VEL
LIN {X 0,Y 357.839,Z 973.644,A -85,B 0,C 180,E1 24145.904,E2 24145.904} C_VEL
LIN {X 0,Y 337.893,Z 1009.06,A -85,B 0,C 180,E1 24149.577,E2 24149.577} C_VEL
LIN {X 0,Y 317.318,Z 1040.107,A -85,B 0,C 180,E1 24154.169,E2 24154.169} C_VEL
LIN {X 0,Y 295.336,Z 1069.051,A -85,B 0,C 180,E1 24160.442,E2 24160.442} C_VEL
LIN {X 0,Y 275.541,Z 1092.867,A -85,B 0,C 180,E1 24168.289,E2 24168.289} C_VEL
LIN {X 0,Y 260.552,Z 1110.773,A -85,B 0,C 180,E1 24177.489,E2 24177.489} C_VEL
LIN {X 0,Y 251.606,Z 1122.359,A -85,B 0,C 180,E1 24187.024,E2 24187.024} C_VEL
LIN {X 0,Y 247.595,Z 1128.413,A -85,B 0,C 180,E1 24195.872,E2 24195.872} C_VEL
LIN {X 0,Y 246.421,Z 1130.687,A -85,B 0,C 180,E1 24206.486,E2 24206.486} C_VEL
LIN {X 0,Y 246.96,Z 1129.264,A -85,B 0,C 180,E1 24213.51,E2 24213.51} C_VEL
LIN {X 0,Y 249.012,Z 1124.02,A -85,B 0,C 180,E1 24222.265,E2 24222.265} C_VEL
LIN {X 0,Y 255.838,Z 1112.655,A -85,B 0,C 180,E1 24232.579,E2 24232.579} C_VEL
LIN {X 0,Y 268.811,Z 1094.471,A -85,B 0,C 180,E1 24242.525,E2 24242.525} C_VEL
LIN {X 0,Y 286.223,Z 1070.949,A -85,B 0,C 180,E1 24250.796,E2 24250.796} C_VEL
LIN {X 0,Y 305.774,Z 1043.175,A -85,B 0,C 180,E1 24257.319,E2 24257.319} C_VEL
LIN {X 0,Y 325.539,Z 1011.726,A -85,B 0,C 180,E1 24262.427,E2 24262.427} C_VEL
LIN {X 0,Y 344.656,Z 976.457,A -85,B 0,C 180,E1 24266.414,E2 24266.414} C_VEL
LIN {X 0,Y 350.037,Z 964.287,A -85,B 0,C 180,E1 24267.609,E2 24267.609} C_VEL
LIN {X 0,Y 348.227,Z 942.714,A -85,B 0,C 180,E1 24272.895,E2 24272.895} C_VEL
LIN {X 0,Y 345.116,Z 924.787,A -85,B 0,C 180,E1 24278.356,E2 24278.356} C_VEL
LIN {X 0,Y 341.388,Z 909.975,A -85,B 0,C 180,E1 24284.597,E2 24284.597} C_VEL
LIN {X 0,Y 338.703,Z 900.579,A -85,B 0,C 180,E1 24290.946,E2 24290.946} C_VEL
LIN {X 0,Y 338.292,Z 896.674,A -85,B 0,C 180,E1 24294.871,E2 24294.871} C_VEL
LIN {X 0,Y 338.495,Z 895.807,A -85,B 0,C 180,E1 24299.996,E2 24299.996} C_VEL
LIN {X 0,Y 340.504,Z 903.078,A -85,B 0,C 180,E1 24307.646,E2 24307.646} C_VEL
LIN {X 0,Y 344.363,Z 914.414,A -85,B 0,C 180,E1 24313.792,E2 24313.792} C_VEL
LIN {X 0,Y 349.084,Z 931.221,A -85,B 0,C 180,E1 24319.823,E2 24319.823} C_VEL
LIN {X 0,Y 352.924,Z 950.782,A -85,B 0,C 180,E1 24325.06,E2 24325.06} C_VEL
LIN {X 0,Y 354.182,Z 963.759,A -85,B 0,C 180,E1 24327.889,E2 24327.889} C_VEL
LIN {X 0,Y 335.011,Z 1003.513,A -85,B 0,C 180,E1 24331.326,E2 24331.326} C_VEL
LIN {X 0,Y 313.483,Z 1040.863,A -85,B 0,C 180,E1 24336.153,E2 24336.153} C_VEL
LIN {X 0,Y 291.555,Z 1074.132,A -85,B 0,C 180,E1 24342.599,E2 24342.599} C_VEL
LIN {X 0,Y 271.921,Z 1102.042,A -85,B 0,C 180,E1 24350.85,E2 24350.85} C_VEL
LIN {X 0,Y 257.836,Z 1122.522,A -85,B 0,C 180,E1 24360.119,E2 24360.119} C_VEL
LIN {X 0,Y 250.012,Z 1136.279,A -85,B 0,C 180,E1 24369.739,E2 24369.739} C_VEL
LIN {X 0,Y 246.87,Z 1144.723,A -85,B 0,C 180,E1 24379.417,E2 24379.417} C_VEL
LIN {X 0,Y 246.51,Z 1147.671,A -85,B 0,C 180,E1 24386.484,E2 24386.484} C_VEL
LIN {X 0,Y 246.762,Z 1148.188,A -85,B 0,C 180,E1 24389.998,E2 24389.998} C_VEL
LIN {X 0,Y 246.502,Z 1147.281,A -85,B 0,C 180,E1 24397.04,E2 24397.04} C_VEL
LIN {X 0,Y 248.119,Z 1142.61,A -85,B 0,C 180,E1 24405.904,E2 24405.904} C_VEL
LIN {X 0,Y 253.728,Z 1132.934,A -85,B 0,C 180,E1 24415.447,E2 24415.447} C_VEL
LIN {X 0,Y 266.196,Z 1116.081,A -85,B 0,C 180,E1 24425.579,E2 24425.579} C_VEL
LIN {X 0,Y 284.756,Z 1092.738,A -85,B 0,C 180,E1 24434.443,E2 24434.443} C_VEL
LIN {X 0,Y 306.53,Z 1064.169,A -85,B 0,C 180,E1 24441.496,E2 24441.496} C_VEL
LIN {X 0,Y 329.293,Z 1031.152,A -85,B 0,C 180,E1 24446.872,E2 24446.872} C_VEL
LIN {X 0,Y 349.781,Z 996.647,A -85,B 0,C 180,E1 24450.704,E2 24450.704} C_VEL
LIN {X 0,Y 363.061,Z 969.772,A -85,B 0,C 180,E1 24453.007,E2 24453.007} C_VEL
LIN {X 0,Y 360.547,Z 950.733,A -85,B 0,C 180,E1 24458.216,E2 24458.216} C_VEL
LIN {X 0,Y 357.299,Z 935.754,A -85,B 0,C 180,E1 24463.653,E2 24463.653} C_VEL
LIN {X 0,Y 354.665,Z 925.565,A -85,B 0,C 180,E1 24468.951,E2 24468.951} C_VEL
LIN {X 0,Y 352.944,Z 918.399,A -85,B 0,C 180,E1 24475.092,E2 24475.092} C_VEL
LIN {X 0,Y 352.487,Z 917.224,A -85,B 0,C 180,E1 24480.004,E2 24480.004} C_VEL
LIN {X 0,Y 352.519,Z 919.362,A -85,B 0,C 180,E1 24483.69,E2 24483.69} C_VEL
LIN {X 0,Y 353.774,Z 927.028,A -85,B 0,C 180,E1 24489.84,E2 24489.84} C_VEL
LIN {X 0,Y 356.035,Z 940.08,A -85,B 0,C 180,E1 24496.015,E2 24496.015} C_VEL
LIN {X 0,Y 357.925,Z 956.086,A -85,B 0,C 180,E1 24501.418,E2 24501.418} C_VEL
LIN {X 0,Y 358.555,Z 969.327,A -85,B 0,C 180,E1 24505.058,E2 24505.058} C_VEL
LIN {X 0,Y 356.271,Z 974.728,A -85,B 0,C 180,E1 24505.654,E2 24505.654} C_VEL
LIN {X 0,Y 346.254,Z 988.563,A -85,B 0,C 180,E1 24506.09,E2 24506.09} C_VEL
LIN {X 0,Y 324.932,Z 1022.883,A -85,B 0,C 180,E1 24510.187,E2 24510.187} C_VEL
LIN {X 0,Y 303.105,Z 1052.975,A -85,B 0,C 180,E1 24515.402,E2 24515.402} C_VEL
LIN {X 0,Y 282.073,Z 1078.764,A -85,B 0,C 180,E1 24521.987,E2 24521.987} C_VEL
LIN {X 0,Y 262.523,Z 1100.97,A -85,B 0,C 180,E1 24530.718,E2 24530.718} C_VEL
LIN {X 0,Y 248.597,Z 1116.98,A -85,B 0,C 180,E1 24540.906,E2 24540.906} C_VEL
LIN {X 0,Y 242.313,Z 1125.107,A -85,B 0,C 180,E1 24549.286,E2 24549.286} C_VEL
LIN {X 0,Y 238.928,Z 1130.035,A -85,B 0,C 180,E1 24559.065,E2 24559.065} C_VEL
LIN {X 0,Y 238.509,Z 1130.974,A -85,B 0,C 180,E1 24566.37,E2 24566.37} C_VEL
LIN {X 0,Y 239.09,Z 1129.562,A -85,B 0,C 180,E1 24573.626,E2 24573.626} C_VEL
LIN {X 0,Y 241.254,Z 1124.349,A -85,B 0,C 180,E1 24582.666,E2 24582.666} C_VEL
LIN {X 0,Y 248.469,Z 1113.013,A -85,B 0,C 180,E1 24593.287,E2 24593.287} C_VEL
LIN {X 0,Y 262.079,Z 1094.86,A -85,B 0,C 180,E1 24603.468,E2 24603.468} C_VEL
LIN {X 0,Y 280.227,Z 1071.376,A -85,B 0,C 180,E1 24611.862,E2 24611.862} C_VEL
LIN {X 0,Y 300.427,Z 1043.647,A -85,B 0,C 180,E1 24618.436,E2 24618.436} C_VEL
LIN {X 0,Y 320.038,Z 1013.474,A -85,B 0,C 180,E1 24623.389,E2 24623.389} C_VEL
LIN {X 0,Y 340.331,Z 977.057,A -85,B 0,C 180,E1 24627.527,E2 24627.527} C_VEL
LIN {X 0,Y 344.59,Z 967.326,A -85,B 0,C 180,E1 24628.529,E2 24628.529} C_VEL
LIN {X 0,Y 343.3,Z 946.464,A -85,B 0,C 180,E1 24633.886,E2 24633.886} C_VEL
LIN {X 0,Y 340.761,Z 929.757,A -85,B 0,C 180,E1 24639.221,E2 24639.221} C_VEL
LIN {X 0,Y 337.792,Z 916.447,A -85,B 0,C 180,E1 24645.093,E2 24645.093} C_VEL
LIN {X 0,Y 335.823,Z 908.049,A -85,B 0,C 180,E1 24650.867,E2 24650.867} C_VEL
LIN {X 0,Y 335.372,Z 904.201,A -85,B 0,C 180,E1 24654.827,E2 24654.827} C_VEL
LIN {X 0,Y 335.611,Z 903.212,A -85,B 0,C 180,E1 24659.996,E2 24659.996} C_VEL
LIN {X 0,Y 337.565,Z 910.693,A -85,B 0,C 180,E1 24667.713,E2 24667.713} C_VEL
LIN {X 0,Y 341.016,Z 922.203,A -85,B 0,C 180,E1 24673.93,E2 24673.93} C_VEL
LIN {X 0,Y 345.078,Z 938.712,A -85,B 0,C 180,E1 24679.831,E2 24679.831} C_VEL
LIN {X 0,Y 348.186,Z 957.613,A -85,B 0,C 180,E1 24684.916,E2 24684.916} C_VEL
LIN {X 0,Y 348.618,Z 967.248,A -85,B 0,C 180,E1 24687.024,E2 24687.024} C_VEL
LIN {X 0,Y 329.636,Z 1005.131,A -85,B 0,C 180,E1 24690.358,E2 24690.358} C_VEL
LIN {X 0,Y 308.754,Z 1040.373,A -85,B 0,C 180,E1 24694.935,E2 24694.935} C_VEL
LIN {X 0,Y 286.921,Z 1072.492,A -85,B 0,C 180,E1 24701.121,E2 24701.121} C_VEL
LIN {X 0,Y 268.03,Z 1098.197,A -85,B 0,C 180,E1 24708.511,E2 24708.511} C_VEL
LIN {X 0,Y 252.879,Z 1118.998,A -85,B 0,C 180,E1 24717.463,E2 24717.463} C_VEL
LIN {X 0,Y 243.532,Z 1133.85,A -85,B 0,C 180,E1 24727.18,E2 24727.18} C_VEL
LIN {X 0,Y 239.236,Z 1143.437,A -85,B 0,C 180,E1 24737.636,E2 24737.636} C_VEL
LIN {X 0,Y 238.596,Z 1147.376,A -85,B 0,C 180,E1 24746.367,E2 24746.367} C_VEL
LIN {X 0,Y 238.857,Z 1147.902,A -85,B 0,C 180,E1 24749.998,E2 24749.998} C_VEL
LIN {X 0,Y 238.61,Z 1147.011,A -85,B 0,C 180,E1 24757.274,E2 24757.274} C_VEL
LIN {X 0,Y 240.402,Z 1142.355,A -85,B 0,C 180,E1 24766.429,E2 24766.429} C_VEL
LIN {X 0,Y 247.009,Z 1131.854,A -85,B 0,C 180,E1 24776.9,E2 24776.9} C_VEL
LIN {X 0,Y 259.595,Z 1115.881,A -85,B 0,C 180,E1 24786.628,E2 24786.628} C_VEL
LIN {X 0,Y 278.465,Z 1093.198,A -85,B 0,C 180,E1 24795.415,E2 24795.415} C_VEL
LIN {X 0,Y 300.379,Z 1065.498,A -85,B 0,C 180,E1 24802.401,E2 24802.401} C_VEL
LIN {X 0,Y 322.36,Z 1034.909,A -85,B 0,C 180,E1 24807.538,E2 24807.538} C_VEL
LIN {X 0,Y 343.838,Z 1000.414,A -85,B 0,C 180,E1 24811.515,E2 24811.515} C_VEL
LIN {X 0,Y 357.509,Z 974.757,A -85,B 0,C 180,E1 24813.68,E2 24813.68} C_VEL
LIN {X 0,Y 356.519,Z 960.059,A -85,B 0,C 180,E1 24817.584,E2 24817.584} C_VEL
LIN {X 0,Y 353.764,Z 943.932,A -85,B 0,C 180,E1 24823.249,E2 24823.249} C_VEL
LIN {X 0,Y 351.153,Z 932.94,A -85,B 0,C 180,E1 24828.839,E2 24828.839} C_VEL
LIN {X 0,Y 349.7,Z 925.745,A -85,B 0,C 180,E1 24835.047,E2 24835.047} C_VEL
LIN {X 0,Y 349.289,Z 924.45,A -85,B 0,C 180,E1 24840.004,E2 24840.004} C_VEL
LIN {X 0,Y 349.157,Z 926.64,A -85,B 0,C 180,E1 24843.725,E2 24843.725} C_VEL
LIN {X 0,Y 350.156,Z 934.411,A -85,B 0,C 180,E1 24849.942,E2 24849.942} C_VEL
LIN {X 0,Y 351.739,Z 946.149,A -85,B 0,C 180,E1 24855.577,E2 24855.577} C_VEL
LIN {X 0,Y 353.1,Z 961.253,A -85,B 0,C 180,E1 24860.841,E2 24860.841} C_VEL
LIN {X 0,Y 353.326,Z 975.018,A -85,B 0,C 180,E1 24864.73,E2 24864.73} C_VEL
LIN {X 0,Y 346.254,Z 988.563,A -85,B 0,C 180,E1 24866.09,E2 24866.09} C_VEL
LIN {X 0,Y 336.379,Z 1002.243,A -85,B 0,C 180,E1 24866.925,E2 24866.925} C_VEL
LIN {X 0,Y 326.191,Z 1015.318,A -85,B 0,C 180,E1 24867.895,E2 24867.895} C_VEL
LIN {X 0,Y 303.32,Z 1046.904,A -85,B 0,C 180,E1 24872.889,E2 24872.889} C_VEL
LIN {X 0,Y 281.748,Z 1072.973,A -85,B 0,C 180,E1 24878.954,E2 24878.954} C_VEL
LIN {X 0,Y 260.924,Z 1096.028,A -85,B 0,C 180,E1 24887.121,E2 24887.121} C_VEL
LIN {X 0,Y 244.545,Z 1113.843,A -85,B 0,C 180,E1 24897.272,E2 24897.272} C_VEL
LIN {X 0,Y 234.742,Z 1125.348,A -85,B 0,C 180,E1 24908.586,E2 24908.586} C_VEL
LIN {X 0,Y 231.091,Z 1130.318,A -85,B 0,C 180,E1 24918.749,E2 24918.749} C_VEL
LIN {X 0,Y 230.597,Z 1131.262,A -85,B 0,C 180,E1 24926.245,E2 24926.245} C_VEL
LIN {X 0,Y 231.202,Z 1129.859,A -85,B 0,C 180,E1 24933.75,E2 24933.75} C_VEL
LIN {X 0,Y 234.267,Z 1123.407,A -85,B 0,C 180,E1 24944.651,E2 24944.651} C_VEL
LIN {X 0,Y 241.964,Z 1112.192,A -85,B 0,C 180,E1 24954.862,E2 24954.862} C_VEL
LIN {X 0,Y 255.597,Z 1095.068,A -85,B 0,C 180,E1 24964.544,E2 24964.544} C_VEL
LIN {X 0,Y 275.295,Z 1070.63,A -85,B 0,C 180,E1 24973.327,E2 24973.327} C_VEL
LIN {X 0,Y 296.316,Z 1042.555,A -85,B 0,C 180,E1 24979.905,E2 24979.905} C_VEL
LIN {X 0,Y 317.359,Z 1010.683,A -85,B 0,C 180,E1 24984.993,E2 24984.993} C_VEL
LIN {X 0,Y 337.089,Z 975.73,A -85,B 0,C 180,E1 24988.843,E2 24988.843} C_VEL
LIN {X 0,Y 339.215,Z 970.689,A -85,B 0,C 180,E1 24989.404,E2 24989.404} C_VEL
LIN {X 0,Y 338.47,Z 950.668,A -85,B 0,C 180,E1 24994.783,E2 24994.783} C_VEL
LIN {X 0,Y 336.366,Z 934.248,A -85,B 0,C 180,E1 25000.311,E2 25000.311} C_VEL
LIN {X 0,Y 333.945,Z 921.792,A -85,B 0,C 180,E1 25006.256,E2 25006.256} C_VEL
LIN {X 0,Y 332.596,Z 915.348,A -85,B 0,C 180,E1 25010.848,E2 25010.848} C_VEL
LIN {X 0,Y 332.488,Z 910.42,A -85,B 0,C 180,E1 25017.392,E2 25017.392} C_VEL
LIN {X 0,Y 332.696,Z 910.608,A -85,B 0,C 180,E1 25019.996,E2 25019.996} C_VEL
LIN {X 0,Y 334.332,Z 918.168,A -85,B 0,C 180,E1 25027.788,E2 25027.788} C_VEL
LIN {X 0,Y 337.325,Z 928.889,A -85,B 0,C 180,E1 25033.596,E2 25033.596} C_VEL
LIN {X 0,Y 340.856,Z 945.506,A -85,B 0,C 180,E1 25039.622,E2 25039.622} C_VEL
LIN {X 0,Y 343.17,Z 963.245,A -85,B 0,C 180,E1 25044.5,E2 25044.5} C_VEL
LIN {X 0,Y 343.212,Z 970.542,A -85,B 0,C 180,E1 25046.113,E2 25046.113} C_VEL
LIN {X 0,Y 323.392,Z 1008.443,A -85,B 0,C 180,E1 25049.549,E2 25049.549} C_VEL
LIN {X 0,Y 302.911,Z 1041.723,A -85,B 0,C 180,E1 25053.964,E2 25053.964} C_VEL
LIN {X 0,Y 280.217,Z 1073.955,A -85,B 0,C 180,E1 25060.31,E2 25060.31} C_VEL
LIN {X 0,Y 259.474,Z 1101.122,A -85,B 0,C 180,E1 25068.511,E2 25068.511} C_VEL
LIN {X 0,Y 243.771,Z 1121.78,A -85,B 0,C 180,E1 25078.201,E2 25078.201} C_VEL
LIN {X 0,Y 234.692,Z 1135.875,A -85,B 0,C 180,E1 25088.623,E2 25088.623} C_VEL
LIN {X 0,Y 231.168,Z 1144.097,A -85,B 0,C 180,E1 25098.689,E2 25098.689} C_VEL
LIN {X 0,Y 230.682,Z 1147.08,A -85,B 0,C 180,E1 25106.242,E2 25106.242} C_VEL
LIN {X 0,Y 230.953,Z 1147.616,A -85,B 0,C 180,E1 25109.998,E2 25109.998} C_VEL
LIN {X 0,Y 230.712,Z 1146.74,A -85,B 0,C 180,E1 25117.525,E2 25117.525} C_VEL
LIN {X 0,Y 232.683,Z 1142.099,A -85,B 0,C 180,E1 25126.99,E2 25126.99} C_VEL
LIN {X 0,Y 239.376,Z 1132.173,A -85,B 0,C 180,E1 25137.353,E2 25137.353} C_VEL
LIN {X 0,Y 253.089,Z 1115.68,A -85,B 0,C 180,E1 25147.731,E2 25147.731} C_VEL
LIN {X 0,Y 273.787,Z 1091.882,A -85,B 0,C 180,E1 25156.993,E2 25156.993} C_VEL
LIN {X 0,Y 297.893,Z 1062.394,A -85,B 0,C 180,E1 25164.252,E2 25164.252} C_VEL
LIN {X 0,Y 322.761,Z 1028.091,A -85,B 0,C 180,E1 25169.676,E2 25169.676} C_VEL
LIN {X 0,Y 345.798,Z 990.296,A -85,B 0,C 180,E1 25173.612,E2 25173.612} C_VEL
LIN {X 0,Y 352.581,Z 977.52,A -85,B 0,C 180,E1 25174.631,E2 25174.631} C_VEL
LIN {X 0,Y 351.092,Z 960.04,A -85,B 0,C 180,E1 25179.867,E2 25179.867} C_VEL
LIN {X 0,Y 348.697,Z 945.974,A -85,B 0,C 180,E1 25185.577,E2 25185.577} C_VEL
LIN {X 0,Y 346.704,Z 936.931,A -85,B 0,C 180,E1 25191.231,E2 25191.231} C_VEL
LIN {X 0,Y 346.148,Z 932.935,A -85,B 0,C 180,E1 25194.996,E2 25194.996} C_VEL
LIN {X 0,Y 345.792,Z 931.518,A -85,B 0,C 180,E1 25200.004,E2 25200.004} C_VEL
LIN {X 0,Y 345.589,Z 933.829,A -85,B 0,C 180,E1 25203.764,E2 25203.764} C_VEL
LIN {X 0,Y 346.349,Z 941.715,A -85,B 0,C 180,E1 25210.053,E2 25210.053} C_VEL
LIN {X 0,Y 347.534,Z 953.743,A -85,B 0,C 180,E1 25215.771,E2 25215.771} C_VEL
LIN {X 0,Y 348.223,Z 968.696,A -85,B 0,C 180,E1 25220.978,E2 25220.978} C_VEL
LIN {X 0,Y 347.611,Z 980.06,A -85,B 0,C 180,E1 25224.095,E2 25224.095} C_VEL
LIN {X 0,Y 326.191,Z 1015.318,A -85,B 0,C 180,E1 25227.895,E2 25227.895} C_VEL
LIN {X 0,Y 315.647,Z 1027.947,A -85,B 0,C 180,E1 25228.991,E2 25228.991} C_VEL
LIN {X 0,Y 304.716,Z 1039.807,A -85,B 0,C 180,E1 25230.257,E2 25230.257} C_VEL
LIN {X 0,Y 280.5,Z 1068.841,A -85,B 0,C 180,E1 25236.448,E2 25236.448} C_VEL
LIN {X 0,Y 259.509,Z 1091.54,A -85,B 0,C 180,E1 25243.908,E2 25243.908} C_VEL
LIN {X 0,Y 242.667,Z 1108.879,A -85,B 0,C 180,E1 25252.62,E2 25252.62} C_VEL
LIN {X 0,Y 230.914,Z 1121.341,A -85,B 0,C 180,E1 25262.739,E2 25262.739} C_VEL
LIN {X 0,Y 225.844,Z 1127.206,A -85,B 0,C 180,E1 25270.457,E2 25270.457} C_VEL
LIN {X 0,Y 222.733,Z 1131.356,A -85,B 0,C 180,E1 25282.204,E2 25282.204} C_VEL
LIN {X 0,Y 223.043,Z 1131.157,A -85,B 0,C 180,E1 25290.002,E2 25290.002} C_VEL
LIN {X 0,Y 224.401,Z 1127.488,A -85,B 0,C 180,E1 25299.694,E2 25299.694} C_VEL
LIN {X 0,Y 230.496,Z 1118.162,A -85,B 0,C 180,E1 25311.138,E2 25311.138} C_VEL
LIN {X 0,Y 242.849,Z 1102.703,A -85,B 0,C 180,E1 25321.934,E2 25321.934} C_VEL
LIN {X 0,Y 260.598,Z 1081.732,A -85,B 0,C 180,E1 25331.081,E2 25331.081} C_VEL
LIN {X 0,Y 281.093,Z 1056.435,A -85,B 0,C 180,E1 25338.275,E2 25338.275} C_VEL
LIN {X 0,Y 302.026,Z 1027.864,A -85,B 0,C 180,E1 25343.784,E2 25343.784} C_VEL
LIN {X 0,Y 324.636,Z 991.808,A -85,B 0,C 180,E1 25348.477,E2 25348.477} C_VEL
LIN {X 0,Y 333.865,Z 974.763,A -85,B 0,C 180,E1 25350.142,E2 25350.142} C_VEL
LIN {X 0,Y 333.57,Z 955.19,A -85,B 0,C 180,E1 25355.583,E2 25355.583} C_VEL
LIN {X 0,Y 331.918,Z 938.878,A -85,B 0,C 180,E1 25361.416,E2 25361.416} C_VEL
LIN {X 0,Y 330.18,Z 928.176,A -85,B 0,C 180,E1 25366.77,E2 25366.77} C_VEL
LIN {X 0,Y 329.071,Z 921.563,A -85,B 0,C 180,E1 25372.079,E2 25372.079} C_VEL
LIN {X 0,Y 329.287,Z 917.66,A -85,B 0,C 180,E1 25377.366,E2 25377.366} C_VEL
LIN {X 0,Y 329.476,Z 917.883,A -85,B 0,C 180,E1 25379.996,E2 25379.996} C_VEL
LIN {X 0,Y 331.057,Z 925.638,A -85,B 0,C 180,E1 25387.865,E2 25387.865} C_VEL
LIN {X 0,Y 333.635,Z 936.517,A -85,B 0,C 180,E1 25393.749,E2 25393.749} C_VEL
LIN {X 0,Y 336.509,Z 952.958,A -85,B 0,C 180,E1 25399.672,E2 25399.672} C_VEL
LIN {X 0,Y 338.167,Z 970.638,A -85,B 0,C 180,E1 25404.539,E2 25404.539} C_VEL
LIN {X 0,Y 337.481,Z 974.744,A -85,B 0,C 180,E1 25405.247,E2 25405.247} C_VEL
LIN {X 0,Y 315.492,Z 1014.698,A -85,B 0,C 180,E1 25409.035,E2 25409.035} C_VEL
LIN {X 0,Y 292.206,Z 1050.16,A -85,B 0,C 180,E1 25414.163,E2 25414.163} C_VEL
LIN {X 0,Y 270.513,Z 1079.098,A -85,B 0,C 180,E1 25420.436,E2 25420.436} C_VEL
LIN {X 0,Y 250.881,Z 1103.741,A -85,B 0,C 180,E1 25428.503,E2 25428.503} C_VEL
LIN {X 0,Y 235.742,Z 1122.927,A -85,B 0,C 180,E1 25438.072,E2 25438.072} C_VEL
LIN {X 0,Y 226.57,Z 1136.667,A -85,B 0,C 180,E1 25448.982,E2 25448.982} C_VEL
LIN {X 0,Y 223.358,Z 1143.783,A -85,B 0,C 180,E1 25458.288,E2 25458.288} C_VEL
LIN {X 0,Y 222.77,Z 1146.785,A -85,B 0,C 180,E1 25466.108,E2 25466.108} C_VEL
LIN {X 0,Y 223.047,Z 1147.331,A -85,B 0,C 180,E1 25469.998,E2 25469.998} C_VEL
LIN {X 0,Y 222.817,Z 1146.469,A -85,B 0,C 180,E1 25477.793,E2 25477.793} C_VEL
LIN {X 0,Y 224.971,Z 1141.842,A -85,B 0,C 180,E1 25487.591,E2 25487.591} C_VEL
LIN {X 0,Y 232.181,Z 1131.943,A -85,B 0,C 180,E1 25498.275,E2 25498.275} C_VEL
LIN {X 0,Y 246.675,Z 1115.48,A -85,B 0,C 180,E1 25508.893,E2 25508.893} C_VEL
LIN {X 0,Y 268.253,Z 1091.717,A -85,B 0,C 180,E1 25518.276,E2 25518.276} C_VEL
LIN {X 0,Y 293.235,Z 1062.273,A -85,B 0,C 180,E1 25525.536,E2 25525.536} C_VEL
LIN {X 0,Y 318.076,Z 1028.974,A -85,B 0,C 180,E1 25530.8,E2 25530.8} C_VEL
LIN {X 0,Y 340.822,Z 992.812,A -85,B 0,C 180,E1 25534.598,E2 25534.598} C_VEL
LIN {X 0,Y 347.283,Z 980.578,A -85,B 0,C 180,E1 25535.697,E2 25535.697} C_VEL
LIN {X 0,Y 346.208,Z 964.08,A -85,B 0,C 180,E1 25540.915,E2 25540.915} C_VEL
LIN {X 0,Y 344.307,Z 950.837,A -85,B 0,C 180,E1 25546.685,E2 25546.685} C_VEL
LIN {X 0,Y 342.756,Z 942.749,A -85,B 0,C 180,E1 25552.405,E2 25552.405} C_VEL
LIN {X 0,Y 342.375,Z 938.793,A -85,B 0,C 180,E1 25557.475,E2 25557.475} C_VEL
LIN {X 0,Y 342.145,Z 939.742,A -85,B 0,C 180,E1 25562.535,E2 25562.535} C_VEL
LIN {X 0,Y 342.286,Z 947.92,A -85,B 0,C 180,E1 25569.532,E2 25569.532} C_VEL
LIN {X 0,Y 343.004,Z 959.641,A -85,B 0,C 180,E1 25575.328,E2 25575.328} C_VEL
LIN {X 0,Y 343.202,Z 974.465,A -85,B 0,C 180,E1 25580.625,E2 25580.625} C_VEL
LIN {X 0,Y 342.85,Z 982.635,A -85,B 0,C 180,E1 25583.089,E2 25583.089} C_VEL
LIN {X 0,Y 320.227,Z 1018.608,A -85,B 0,C 180,E1 25587.044,E2 25587.044} C_VEL
LIN {X 0,Y 304.716,Z 1039.807,A -85,B 0,C 180,E1 25590.257,E2 25590.257} C_VEL
LIN {X 0,Y 293.606,Z 1051.166,A -85,B 0,C 180,E1 25591.684,E2 25591.684} C_VEL
LIN {X 0,Y 282.318,Z 1061.788,A -85,B 0,C 180,E1 25593.303,E2 25593.303} C_VEL
LIN {X 0,Y 257.852,Z 1087.84,A -85,B 0,C 180,E1 25601.02,E2 25601.02} C_VEL
LIN {X 0,Y 237.653,Z 1107.658,A -85,B 0,C 180,E1 25610.52,E2 25610.52} C_VEL
LIN {X 0,Y 224.181,Z 1121.013,A -85,B 0,C 180,E1 25621.19,E2 25621.19} C_VEL
LIN {X 0,Y 218.244,Z 1127.458,A -85,B 0,C 180,E1 25629.748,E2 25629.748} C_VEL
LIN {X 0,Y 214.844,Z 1131.634,A -85,B 0,C 180,E1 25641.916,E2 25641.916} C_VEL
LIN {X 0,Y 215.137,Z 1131.453,A -85,B 0,C 180,E1 25650.002,E2 25650.002} C_VEL
LIN {X 0,Y 216.6,Z 1127.805,A -85,B 0,C 180,E1 25660.047,E2 25660.047} C_VEL
LIN {X 0,Y 223.081,Z 1118.511,A -85,B 0,C 180,E1 25671.876,E2 25671.876} C_VEL
LIN {X 0,Y 236.117,Z 1103.078,A -85,B 0,C 180,E1 25682.958,E2 25682.958} C_VEL
LIN {X 0,Y 254.641,Z 1082.143,A -85,B 0,C 180,E1 25692.26,E2 25692.26} C_VEL
LIN {X 0,Y 275.086,Z 1057.866,A -85,B 0,C 180,E1 25699.284,E2 25699.284} C_VEL
LIN {X 0,Y 297.392,Z 1028.369,A -85,B 0,C 180,E1 25705.022,E2 25705.022} C_VEL
LIN {X 0,Y 321.048,Z 991.577,A -85,B 0,C 180,E1 25709.765,E2 25709.765} C_VEL
LIN {X 0,Y 328.625,Z 977.47,A -85,B 0,C 180,E1 25711.256,E2 25711.256} C_VEL
LIN {X 0,Y 328.651,Z 958.337,A -85,B 0,C 180,E1 25716.868,E2 25716.868} C_VEL
LIN {X 0,Y 327.474,Z 943.288,A -85,B 0,C 180,E1 25722.626,E2 25722.626} C_VEL
LIN {X 0,Y 326.167,Z 933.127,A -85,B 0,C 180,E1 25728.282,E2 25728.282} C_VEL
LIN {X 0,Y 325.738,Z 926.369,A -85,B 0,C 180,E1 25734.673,E2 25734.673} C_VEL
LIN {X 0,Y 326.069,Z 924.916,A -85,B 0,C 180,E1 25737.34,E2 25737.34} C_VEL
LIN {X 0,Y 326.26,Z 925.144,A -85,B 0,C 180,E1 25739.996,E2 25739.996} C_VEL
LIN {X 0,Y 327.144,Z 931.115,A -85,B 0,C 180,E1 25746.626,E2 25746.626} C_VEL
LIN {X 0,Y 329.318,Z 941.439,A -85,B 0,C 180,E1 25752.657,E2 25752.657} C_VEL
LIN {X 0,Y 331.677,Z 956.838,A -85,B 0,C 180,E1 25758.59,E2 25758.59} C_VEL
LIN {X 0,Y 332.966,Z 974.656,A -85,B 0,C 180,E1 25763.728,E2 25763.728} C_VEL
LIN {X 0,Y 332.493,Z 977.258,A -85,B 0,C 180,E1 25764.242,E2 25764.242} C_VEL
LIN {X 0,Y 310.431,Z 1016.083,A -85,B 0,C 180,E1 25767.949,E2 25767.949} C_VEL
LIN {X 0,Y 286.401,Z 1051.522,A -85,B 0,C 180,E1 25773.134,E2 25773.134} C_VEL
LIN {X 0,Y 261.758,Z 1083.065,A -85,B 0,C 180,E1 25780.267,E2 25780.267} C_VEL
LIN {X 0,Y 240.278,Z 1108.725,A -85,B 0,C 180,E1 25789.512,E2 25789.512} C_VEL
LIN {X 0,Y 225.838,Z 1126.361,A -85,B 0,C 180,E1 25799.602,E2 25799.602} C_VEL
LIN {X 0,Y 218.201,Z 1137.739,A -85,B 0,C 180,E1 25809.739,E2 25809.739} C_VEL
LIN {X 0,Y 215.197,Z 1144.174,A -85,B 0,C 180,E1 25819.358,E2 25819.358} C_VEL
LIN {X 0,Y 215.142,Z 1147.045,A -85,B 0,C 180,E1 25829.998,E2 25829.998} C_VEL
LIN {X 0,Y 215.228,Z 1145.479,A -85,B 0,C 180,E1 25840.686,E2 25840.686} C_VEL
LIN {X 0,Y 219.141,Z 1138.92,A -85,B 0,C 180,E1 25851.869,E2 25851.869} C_VEL
LIN {X 0,Y 229.216,Z 1127.052,A -85,B 0,C 180,E1 25862.946,E2 25862.946} C_VEL
LIN {X 0,Y 247.124,Z 1108.221,A -85,B 0,C 180,E1 25873.462,E2 25873.462} C_VEL
LIN {X 0,Y 271.097,Z 1082.574,A -85,B 0,C 180,E1 25882.197,E2 25882.197} C_VEL
LIN {X 0,Y 296.512,Z 1052.52,A -85,B 0,C 180,E1 25888.605,E2 25888.605} C_VEL
LIN {X 0,Y 321.304,Z 1018.518,A -85,B 0,C 180,E1 25893.323,E2 25893.323} C_VEL
LIN {X 0,Y 342.093,Z 984.394,A -85,B 0,C 180,E1 25896.583,E2 25896.583} C_VEL
LIN {X 0,Y 341.396,Z 968.296,A -85,B 0,C 180,E1 25901.958,E2 25901.958} C_VEL
LIN {X 0,Y 339.947,Z 955.639,A -85,B 0,C 180,E1 25907.932,E2 25907.932} C_VEL
LIN {X 0,Y 338.725,Z 947.194,A -85,B 0,C 180,E1 25914.886,E2 25914.886} C_VEL
LIN {X 0,Y 338.489,Z 945.542,A -85,B 0,C 180,E1 25920.004,E2 25920.004} C_VEL
LIN {X 0,Y 337.998,Z 949.239,A -85,B 0,C 180,E1 25925.133,E2 25925.133} C_VEL
LIN {X 0,Y 338.272,Z 956.754,A -85,B 0,C 180,E1 25930.66,E2 25930.66} C_VEL
LIN {X 0,Y 338.44,Z 970.44,A -85,B 0,C 180,E1 25936.872,E2 25936.872} C_VEL
LIN {X 0,Y 337.702,Z 985.555,A -85,B 0,C 180,E1 25941.962,E2 25941.962} C_VEL
LIN {X 0,Y 332.382,Z 994.923,A -85,B 0,C 180,E1 25942.998,E2 25942.998} C_VEL
LIN {X 0,Y 308.303,Z 1030.044,A -85,B 0,C 180,E1 25947.334,E2 25947.334} C_VEL
LIN {X 0,Y 282.318,Z 1061.788,A -85,B 0,C 180,E1 25953.303,E2 25953.303} C_VEL
LIN {X 0,Y 270.926,Z 1071.787,A -85,B 0,C 180,E1 25955.135,E2 25955.135} C_VEL
LIN {X 0,Y 259.562,Z 1081.061,A -85,B 0,C 180,E1 25957.19,E2 25957.19} C_VEL
LIN {X 0,Y 237.993,Z 1101.717,A -85,B 0,C 180,E1 25965.702,E2 25965.702} C_VEL
LIN {X 0,Y 222.312,Z 1116.267,A -85,B 0,C 180,E1 25975.39,E2 25975.39} C_VEL
LIN {X 0,Y 211.693,Z 1126.666,A -85,B 0,C 180,E1 25987.108,E2 25987.108} C_VEL
LIN {X 0,Y 207.599,Z 1131.112,A -85,B 0,C 180,E1 25997.389,E2 25997.389} C_VEL
LIN {X 0,Y 206.88,Z 1132.123,A -85,B 0,C 180,E1 26005.814,E2 26005.814} C_VEL
LIN {X 0,Y 207.552,Z 1130.748,A -85,B 0,C 180,E1 26014.178,E2 26014.178} C_VEL
LIN {X 0,Y 210.429,Z 1125.601,A -85,B 0,C 180,E1 26024.649,E2 26024.649} C_VEL
LIN {X 0,Y 219.224,Z 1114.691,A -85,B 0,C 180,E1 26036.358,E2 26036.358} C_VEL
LIN {X 0,Y 234,Z 1098.53,A -85,B 0,C 180,E1 26046.682,E2 26046.682} C_VEL
LIN {X 0,Y 253.15,Z 1077.774,A -85,B 0,C 180,E1 26055.143,E2 26055.143} C_VEL
LIN {X 0,Y 276.646,Z 1050.23,A -85,B 0,C 180,E1 26062.378,E2 26062.378} C_VEL
LIN {X 0,Y 301.524,Z 1016.613,A -85,B 0,C 180,E1 26068.088,E2 26068.088} C_VEL
LIN {X 0,Y 323.323,Z 981.077,A -85,B 0,C 180,E1 26072.137,E2 26072.137} C_VEL
LIN {X 0,Y 323.901,Z 962.995,A -85,B 0,C 180,E1 26077.693,E2 26077.693} C_VEL
LIN {X 0,Y 323.291,Z 949.589,A -85,B 0,C 180,E1 26083.013,E2 26083.013} C_VEL
LIN {X 0,Y 322.359,Z 939.048,A -85,B 0,C 180,E1 26089.19,E2 26089.19} C_VEL
LIN {X 0,Y 322.16,Z 933.587,A -85,B 0,C 180,E1 26094.614,E2 26094.614} C_VEL
LIN {X 0,Y 322.539,Z 932.026,A -85,B 0,C 180,E1 26097.311,E2 26097.311} C_VEL
LIN {X 0,Y 322.728,Z 932.271,A -85,B 0,C 180,E1 26099.996,E2 26099.996} C_VEL
LIN {X 0,Y 323.535,Z 938.414,A -85,B 0,C 180,E1 26106.7,E2 26106.7} C_VEL
LIN {X 0,Y 325.321,Z 948.712,A -85,B 0,C 180,E1 26112.717,E2 26112.717} C_VEL
LIN {X 0,Y 327.074,Z 963.746,A -85,B 0,C 180,E1 26118.512,E2 26118.512} C_VEL
LIN {X 0,Y 327.684,Z 979.151,A -85,B 0,C 180,E1 26123.067,E2 26123.067} C_VEL
LIN {X 0,Y 306.284,Z 1016.207,A -85,B 0,C 180,E1 26126.686,E2 26126.686} C_VEL
LIN {X 0,Y 281.335,Z 1051.925,A -85,B 0,C 180,E1 26131.901,E2 26131.901} C_VEL
LIN {X 0,Y 256.386,Z 1082.833,A -85,B 0,C 180,E1 26138.929,E2 26138.929} C_VEL
LIN {X 0,Y 234.087,Z 1108.337,A -85,B 0,C 180,E1 26148.206,E2 26148.206} C_VEL
LIN {X 0,Y 218.548,Z 1126.339,A -85,B 0,C 180,E1 26158.761,E2 26158.761} C_VEL
LIN {X 0,Y 210.613,Z 1137.41,A -85,B 0,C 180,E1 26168.975,E2 26168.975} C_VEL
LIN {X 0,Y 207.679,Z 1143.15,A -85,B 0,C 180,E1 26177.389,E2 26177.389} C_VEL
LIN {X 0,Y 206.949,Z 1146.195,A -85,B 0,C 180,E1 26185.81,E2 26185.81} C_VEL
LIN {X 0,Y 207.235,Z 1146.759,A -85,B 0,C 180,E1 26189.998,E2 26189.998} C_VEL
LIN {X 0,Y 207.067,Z 1145.929,A -85,B 0,C 180,E1 26198.39,E2 26198.39} C_VEL
LIN {X 0,Y 209.652,Z 1141.33,A -85,B 0,C 180,E1 26208.923,E2 26208.923} C_VEL
LIN {X 0,Y 217.868,Z 1131.558,A -85,B 0,C 180,E1 26220.246,E2 26220.246} C_VEL
LIN {X 0,Y 233.717,Z 1115.494,A -85,B 0,C 180,E1 26231.183,E2 26231.183} C_VEL
LIN {X 0,Y 256.55,Z 1092.493,A -85,B 0,C 180,E1 26240.628,E2 26240.628} C_VEL
LIN {X 0,Y 282.293,Z 1064.355,A -85,B 0,C 180,E1 26247.76,E2 26247.76} C_VEL
LIN {X 0,Y 306.254,Z 1034.572,A -85,B 0,C 180,E1 26252.638,E2 26252.638} C_VEL
LIN {X 0,Y 329.738,Z 1000.342,A -85,B 0,C 180,E1 26256.423,E2 26256.423} C_VEL
LIN {X 0,Y 336.53,Z 989.093,A -85,B 0,C 180,E1 26257.374,E2 26257.374} C_VEL
LIN {X 0,Y 336.846,Z 977.63,A -85,B 0,C 180,E1 26261.028,E2 26261.028} C_VEL
LIN {X 0,Y 335.953,Z 965.444,A -85,B 0,C 180,E1 26266.347,E2 26266.347} C_VEL
LIN {X 0,Y 335.152,Z 958.306,A -85,B 0,C 180,E1 26270.926,E2 26270.926} C_VEL
LIN {X 0,Y 334.838,Z 954.224,A -85,B 0,C 180,E1 26274.826,E2 26274.826} C_VEL
LIN {X 0,Y 334.649,Z 952.459,A -85,B 0,C 180,E1 26280.004,E2 26280.004} C_VEL
LIN {X 0,Y 333.97,Z 956.511,A -85,B 0,C 180,E1 26285.498,E2 26285.498} C_VEL
LIN {X 0,Y 333.934,Z 963.924,A -85,B 0,C 180,E1 26290.8,E2 26290.8} C_VEL
LIN {X 0,Y 333.616,Z 976.282,A -85,B 0,C 180,E1 26296.493,E2 26296.493} C_VEL
LIN {X 0,Y 332.208,Z 990.395,A -85,B 0,C 180,E1 26301.275,E2 26301.275} C_VEL
LIN {X 0,Y 308.874,Z 1024.465,A -85,B 0,C 180,E1 26305.171,E2 26305.171} C_VEL
LIN {X 0,Y 285.251,Z 1053.613,A -85,B 0,C 180,E1 26310.079,E2 26310.079} C_VEL
LIN {X 0,Y 259.991,Z 1080.654,A -85,B 0,C 180,E1 26317.053,E2 26317.053} C_VEL
LIN {X 0,Y 259.562,Z 1081.061,A -85,B 0,C 180,E1 26317.19,E2 26317.19} C_VEL
LIN {X 0,Y 248.247,Z 1089.669,A -85,B 0,C 180,E1 26319.521,E2 26319.521} C_VEL
LIN {X 0,Y 237.066,Z 1097.542,A -85,B 0,C 180,E1 26322.117,E2 26322.117} C_VEL
LIN {X 0,Y 217.118,Z 1115.213,A -85,B 0,C 180,E1 26333.027,E2 26333.027} C_VEL
LIN {X 0,Y 205.879,Z 1125.322,A -85,B 0,C 180,E1 26343.874,E2 26343.874} C_VEL
LIN {X 0,Y 201.126,Z 1129.975,A -85,B 0,C 180,E1 26352.513,E2 26352.513} C_VEL
LIN {X 0,Y 199.102,Z 1132.19,A -85,B 0,C 180,E1 26361.272,E2 26361.272} C_VEL
LIN {X 0,Y 199.321,Z 1132.041,A -85,B 0,C 180,E1 26370.002,E2 26370.002} C_VEL
LIN {X 0,Y 201.027,Z 1128.44,A -85,B 0,C 180,E1 26380.834,E2 26380.834} C_VEL
LIN {X 0,Y 208.38,Z 1119.203,A -85,B 0,C 180,E1 26393.508,E2 26393.508} C_VEL
LIN {X 0,Y 223.748,Z 1102.967,A -85,B 0,C 180,E1 26405.723,E2 26405.723} C_VEL
LIN {X 0,Y 245.459,Z 1080.487,A -85,B 0,C 180,E1 26415.7,E2 26415.7} C_VEL
LIN {X 0,Y 269.388,Z 1053.606,A -85,B 0,C 180,E1 26423.07,E2 26423.07} C_VEL
LIN {X 0,Y 292.587,Z 1023.742,A -85,B 0,C 180,E1 26428.451,E2 26428.451} C_VEL
LIN {X 0,Y 315.421,Z 989.229,A -85,B 0,C 180,E1 26432.607,E2 26432.607} C_VEL
LIN {X 0,Y 318.132,Z 984.219,A -85,B 0,C 180,E1 26433.173,E2 26433.173} C_VEL
LIN {X 0,Y 319.118,Z 967.326,A -85,B 0,C 180,E1 26438.642,E2 26438.642} C_VEL
LIN {X 0,Y 318.883,Z 954.264,A -85,B 0,C 180,E1 26444.187,E2 26444.187} C_VEL
LIN {X 0,Y 318.388,Z 944.494,A -85,B 0,C 180,E1 26450.434,E2 26450.434} C_VEL
LIN {X 0,Y 319,Z 939.143,A -85,B 0,C 180,E1 26457.281,E2 26457.281} C_VEL
LIN {X 0,Y 319.111,Z 940.376,A -85,B 0,C 180,E1 26461.352,E2 26461.352} C_VEL
LIN {X 0,Y 320.042,Z 947.498,A -85,B 0,C 180,E1 26468.138,E2 26468.138} C_VEL
LIN {X 0,Y 321.436,Z 957.835,A -85,B 0,C 180,E1 26473.588,E2 26473.588} C_VEL
LIN {X 0,Y 322.526,Z 973.893,A -85,B 0,C 180,E1 26479.493,E2 26479.493} C_VEL
LIN {X 0,Y 322.409,Z 983.054,A -85,B 0,C 180,E1 26482.203,E2 26482.203} C_VEL
LIN {X 0,Y 300.731,Z 1018.625,A -85,B 0,C 180,E1 26485.664,E2 26485.664} C_VEL
LIN {X 0,Y 276.388,Z 1052.349,A -85,B 0,C 180,E1 26490.634,E2 26490.634} C_VEL
LIN {X 0,Y 250.85,Z 1082.898,A -85,B 0,C 180,E1 26497.616,E2 26497.616} C_VEL
LIN {X 0,Y 228.35,Z 1107.631,A -85,B 0,C 180,E1 26506.694,E2 26506.694} C_VEL
LIN {X 0,Y 211.589,Z 1125.977,A -85,B 0,C 180,E1 26517.611,E2 26517.611} C_VEL
LIN {X 0,Y 203.073,Z 1137.081,A -85,B 0,C 180,E1 26528.155,E2 26528.155} C_VEL
LIN {X 0,Y 199.244,Z 1144.286,A -85,B 0,C 180,E1 26540.284,E2 26540.284} C_VEL
LIN {X 0,Y 199.328,Z 1146.474,A -85,B 0,C 180,E1 26549.998,E2 26549.998} C_VEL
LIN {X 0,Y 199.255,Z 1145.403,A -85,B 0,C 180,E1 26559.733,E2 26559.733} C_VEL
LIN {X 0,Y 203.152,Z 1139.728,A -85,B 0,C 180,E1 26571.831,E2 26571.831} C_VEL
LIN {X 0,Y 214.373,Z 1127.86,A -85,B 0,C 180,E1 26584.324,E2 26584.324} C_VEL
LIN {X 0,Y 231.489,Z 1111.524,A -85,B 0,C 180,E1 26594.438,E2 26594.438} C_VEL
LIN {X 0,Y 254.564,Z 1089.234,A -85,B 0,C 180,E1 26603.007,E2 26603.007} C_VEL
LIN {X 0,Y 280.204,Z 1061.894,A -85,B 0,C 180,E1 26609.635,E2 26609.635} C_VEL
LIN {X 0,Y 308.148,Z 1027.174,A -85,B 0,C 180,E1 26614.957,E2 26614.957} C_VEL
LIN {X 0,Y 331.771,Z 991.911,A -85,B 0,C 180,E1 26618.416,E2 26618.416} C_VEL
LIN {X 0,Y 331.795,Z 976.737,A -85,B 0,C 180,E1 26624.149,E2 26624.149} C_VEL
LIN {X 0,Y 331.151,Z 966.965,A -85,B 0,C 180,E1 26629.489,E2 26629.489} C_VEL
LIN {X 0,Y 330.705,Z 961.111,A -85,B 0,C 180,E1 26634.762,E2 26634.762} C_VEL
LIN {X 0,Y 330.585,Z 959.273,A -85,B 0,C 180,E1 26640.004,E2 26640.004} C_VEL
LIN {X 0,Y 329.792,Z 963.044,A -85,B 0,C 180,E1 26645.261,E2 26645.261} C_VEL
LIN {X 0,Y 329.368,Z 971.514,A -85,B 0,C 180,E1 26651.246,E2 26651.246} C_VEL
LIN {X 0,Y 328.573,Z 983.614,A -85,B 0,C 180,E1 26656.754,E2 26656.754} C_VEL
LIN {X 0,Y 327.017,Z 994.059,A -85,B 0,C 180,E1 26660.302,E2 26660.302} C_VEL
LIN {X 0,Y 302.449,Z 1028.571,A -85,B 0,C 180,E1 26664.347,E2 26664.347} C_VEL
LIN {X 0,Y 276.343,Z 1059.064,A -85,B 0,C 180,E1 26669.768,E2 26669.768} C_VEL
LIN {X 0,Y 252.486,Z 1083.269,A -85,B 0,C 180,E1 26676.42,E2 26676.42} C_VEL
LIN {X 0,Y 237.066,Z 1097.542,A -85,B 0,C 180,E1 26682.117,E2 26682.117} C_VEL
LIN {X 0,Y 226.162,Z 1104.684,A -85,B 0,C 180,E1 26685.036,E2 26685.036} C_VEL
LIN {X 0,Y 215.852,Z 1111.033,A -85,B 0,C 180,E1 26688.317,E2 26688.317} C_VEL
LIN {X 0,Y 201.566,Z 1123.036,A -85,B 0,C 180,E1 26699.377,E2 26699.377} C_VEL
LIN {X 0,Y 193.457,Z 1130.236,A -85,B 0,C 180,E1 26711.796,E2 26711.796} C_VEL
LIN {X 0,Y 191.243,Z 1132.468,A -85,B 0,C 180,E1 26720.91,E2 26720.91} C_VEL
LIN {X 0,Y 191.418,Z 1132.333,A -85,B 0,C 180,E1 26730.003,E2 26730.003} C_VEL
LIN {X 0,Y 193.232,Z 1128.813,A -85,B 0,C 180,E1 26741.165,E2 26741.165} C_VEL
LIN {X 0,Y 201.073,Z 1119.547,A -85,B 0,C 180,E1 26754.417,E2 26754.417} C_VEL
LIN {X 0,Y 217.307,Z 1103.342,A -85,B 0,C 180,E1 26766.954,E2 26766.954} C_VEL
LIN {X 0,Y 239.955,Z 1080.898,A -85,B 0,C 180,E1 26777.064,E2 26777.064} C_VEL
LIN {X 0,Y 264.552,Z 1054.185,A -85,B 0,C 180,E1 26784.425,E2 26784.425} C_VEL
LIN {X 0,Y 287.871,Z 1025.117,A -85,B 0,C 180,E1 26789.668,E2 26789.668} C_VEL
LIN {X 0,Y 311.5,Z 990.404,A -85,B 0,C 180,E1 26793.841,E2 26793.841} C_VEL
LIN {X 0,Y 312.986,Z 987.432,A -85,B 0,C 180,E1 26794.245,E2 26794.245} C_VEL
LIN {X 0,Y 314.313,Z 971.648,A -85,B 0,C 180,E1 26799.6,E2 26799.6} C_VEL
LIN {X 0,Y 314.476,Z 958.939,A -85,B 0,C 180,E1 26805.386,E2 26805.386} C_VEL
LIN {X 0,Y 314.411,Z 950.228,A -85,B 0,C 180,E1 26811.707,E2 26811.707} C_VEL
LIN {X 0,Y 315.166,Z 946.132,A -85,B 0,C 180,E1 26817.248,E2 26817.248} C_VEL
LIN {X 0,Y 315.269,Z 947.331,A -85,B 0,C 180,E1 26821.369,E2 26821.369} C_VEL
LIN {X 0,Y 316.097,Z 954.669,A -85,B 0,C 180,E1 26828.24,E2 26828.24} C_VEL
LIN {X 0,Y 316.993,Z 965.267,A -85,B 0,C 180,E1 26833.782,E2 26833.782} C_VEL
LIN {X 0,Y 317.45,Z 980.681,A -85,B 0,C 180,E1 26839.456,E2 26839.456} C_VEL
LIN {X 0,Y 317.238,Z 986.5,A -85,B 0,C 180,E1 26841.184,E2 26841.184} C_VEL
LIN {X 0,Y 293.635,Z 1023.444,A -85,B 0,C 180,E1 26844.9,E2 26844.9} C_VEL
LIN {X 0,Y 269.739,Z 1054.985,A -85,B 0,C 180,E1 26849.735,E2 26849.735} C_VEL
LIN {X 0,Y 245.787,Z 1082.655,A -85,B 0,C 180,E1 26856.163,E2 26856.163} C_VEL
LIN {X 0,Y 222.472,Z 1107.237,A -85,B 0,C 180,E1 26865.25,E2 26865.25} C_VEL
LIN {X 0,Y 204.741,Z 1125.616,A -85,B 0,C 180,E1 26876.387,E2 26876.387} C_VEL
LIN {X 0,Y 194.953,Z 1137.578,A -85,B 0,C 180,E1 26888.412,E2 26888.412} C_VEL
LIN {X 0,Y 191.302,Z 1144.382,A -85,B 0,C 180,E1 26900.908,E2 26900.908} C_VEL
LIN {X 0,Y 191.423,Z 1146.188,A -85,B 0,C 180,E1 26909.997,E2 26909.997} C_VEL
LIN {X 0,Y 191.31,Z 1145.388,A -85,B 0,C 180,E1 26919.087,E2 26919.087} C_VEL
LIN {X 0,Y 195.046,Z 1140.15,A -85,B 0,C 180,E1 26931.656,E2 26931.656} C_VEL
LIN {X 0,Y 206.353,Z 1128.807,A -85,B 0,C 180,E1 26944.575,E2 26944.575} C_VEL
LIN {X 0,Y 224.204,Z 1112.722,A -85,B 0,C 180,E1 26955.197,E2 26955.197} C_VEL
LIN {X 0,Y 247.348,Z 1091.416,A -85,B 0,C 180,E1 26963.791,E2 26963.791} C_VEL
LIN {X 0,Y 274.41,Z 1063.66,A -85,B 0,C 180,E1 26970.708,E2 26970.708} C_VEL
LIN {X 0,Y 300.412,Z 1032.798,A -85,B 0,C 180,E1 26975.596,E2 26975.596} C_VEL
LIN {X 0,Y 325.331,Z 997.595,A -85,B 0,C 180,E1 26979.257,E2 26979.257} C_VEL
LIN {X 0,Y 326.651,Z 994.754,A -85,B 0,C 180,E1 26979.703,E2 26979.703} C_VEL
LIN {X 0,Y 326.973,Z 981.063,A -85,B 0,C 180,E1 26985.283,E2 26985.283} C_VEL
LIN {X 0,Y 326.652,Z 972.158,A -85,B 0,C 180,E1 26990.688,E2 26990.688} C_VEL
LIN {X 0,Y 326.551,Z 966.281,A -85,B 0,C 180,E1 26997.352,E2 26997.352} C_VEL
LIN {X 0,Y 326.43,Z 966.021,A -85,B 0,C 180,E1 27000.004,E2 27000.004} C_VEL
LIN {X 0,Y 325.475,Z 969.881,A -85,B 0,C 180,E1 27005.331,E2 27005.331} C_VEL
LIN {X 0,Y 324.773,Z 977.302,A -85,B 0,C 180,E1 27010.728,E2 27010.728} C_VEL
LIN {X 0,Y 323.526,Z 989.045,A -85,B 0,C 180,E1 27016.276,E2 27016.276} C_VEL
LIN {X 0,Y 321.63,Z 997.994,A -85,B 0,C 180,E1 27019.339,E2 27019.339} C_VEL
LIN {X 0,Y 297.657,Z 1030.57,A -85,B 0,C 180,E1 27023.205,E2 27023.205} C_VEL
LIN {X 0,Y 269.731,Z 1062.071,A -85,B 0,C 180,E1 27028.917,E2 27028.917} C_VEL
LIN {X 0,Y 242.415,Z 1088.327,A -85,B 0,C 180,E1 27036.627,E2 27036.627} C_VEL
LIN {X 0,Y 219.229,Z 1108.255,A -85,B 0,C 180,E1 27046.43,E2 27046.43} C_VEL
LIN {X 0,Y 215.852,Z 1111.033,A -85,B 0,C 180,E1 27048.317,E2 27048.317} C_VEL
LIN {X 0,Y 206.003,Z 1116.627,A -85,B 0,C 180,E1 27051.962,E2 27051.962} C_VEL
LIN {X 0,Y 196.821,Z 1121.44,A -85,B 0,C 180,E1 27055.996,E2 27055.996} C_VEL
LIN {X 0,Y 187.312,Z 1129.233,A -85,B 0,C 180,E1 27067.874,E2 27067.874} C_VEL
LIN {X 0,Y 183.377,Z 1132.747,A -85,B 0,C 180,E1 27080.517,E2 27080.517} C_VEL
LIN {X 0,Y 183.508,Z 1132.622,A -85,B 0,C 180,E1 27090.003,E2 27090.003} C_VEL
LIN {X 0,Y 185.748,Z 1128.687,A -85,B 0,C 180,E1 27102.529,E2 27102.529} C_VEL
LIN {X 0,Y 193.842,Z 1119.888,A -85,B 0,C 180,E1 27115.391,E2 27115.391} C_VEL
LIN {X 0,Y 211.235,Z 1103.487,A -85,B 0,C 180,E1 27128.404,E2 27128.404} C_VEL
LIN {X 0,Y 234.576,Z 1081.309,A -85,B 0,C 180,E1 27138.495,E2 27138.495} C_VEL
LIN {X 0,Y 259.689,Z 1054.969,A -85,B 0,C 180,E1 27145.782,E2 27145.782} C_VEL
LIN {X 0,Y 284.439,Z 1024.952,A -85,B 0,C 180,E1 27151.151,E2 27151.151} C_VEL
LIN {X 0,Y 307.493,Z 991.983,A -85,B 0,C 180,E1 27155.064,E2 27155.064} C_VEL
